        // Force cleanup of all IO bytes and explicit triggers on failure
        GVL.Robot.ACK_Complete     := 0;
        GVL.Robot.CMD              := 0;
        
        IF NOT xExecute THEN
            iHandshakeState := 0;
        END_IF;

END_CASE;

END_FUNCTION_BLOCK

// Device/Application/F002_PART_X/F002_SR01_SOCKET_SERVER
PROGRAM F002_SR01_SOCKET_SERVER
VAR
    ipAddr : NBS.IP_ADDR := (sAddr:= '192.168.0.247');
	Server: NBS.TCP_Server :=(uiPort :=2000);
	

	Connection: NBS.TCP_Connection;
	Read : NBS.TCP_Read;
	Write : NBS.TCP_Write;
	
	T1: TON := (PT := TIME#50MS);
	xEnableServer: BOOL;
	
	ReadData: ARRAY[0..3] OF DINT;
END_VAR
VAR_INPUT
	WriteData:  ARRAY[0..9] OF BYTE;
END_VAR

//TCP Sockets Server

//Server Instance
Server(xEnable:=GVL.PARTX.ENABLE_TCP,
		ipAddr:= ipAddr
		);
		
//Conection INstance	
Connection(xEnable:=(Server.xbusy AND NOT(Connection.xDone)),
		hServer:= Server.hServer
		);
		
//Read Data		
Read(xEnable:= Connection.xActive,
		hConnection:=Connection.hConnection,
		szSize:=SIZEOF(ReadData),
		pData:=ADR(ReadData)
		);

		
//Write Data	
Write(xExecute:= Connection.xActive AND T1.Q,
		hConnection:=Connection.hConnection,
		szSize:=SIZEOF(WriteData),
		pData:=ADR(WriteData)
		);

//Write Data Time Interval	
T1(IN:=NOT(Write.xDone));

END_PROGRAM

// Device/Application/F002_PART_X/F002_SR02_SOCKET_CLIENT
PROGRAM F002_SR02_SOCKET_CLIENT
VAR
    ipAddr : NBS.IP_ADDR := (sAddr:= '192.168.1.11');
	Client: NBS.TCP_Client :=(uiPort :=2000);
	

	Connection: NBS.TCP_Connection;
	Read : NBS.TCP_Read;
	Write : NBS.TCP_Write;
	
	T1: TON := (PT := TIME#50MS);
	xEnableServer: BOOL;
	
	ReadData: ARRAY[0..3] OF DINT;
END_VAR
VAR_INPUT
	WriteData:  ARRAY[0..9] OF BYTE;
END_VAR

//TCP Sockets Client

//Client Instance
Client(xEnable:=GVL.PARTX.ENABLE_TCP,
		ipAddr:= ipAddr
		);
		
		
//Read Data		
Read(xEnable:= Client.xActive,
		hConnection:=Client.hConnection,
		szSize:=SIZEOF(ReadData),
		pData:=ADR(ReadData)
		);

		
//Write Data	
Write(xExecute:= Client.xActive AND T1.Q,
		hConnection:=Client.hConnection,
		szSize:=SIZEOF(WriteData),
		pData:=ADR(WriteData)
		);

//Write Data Time Interval	
T1(IN:=NOT(Write.xDone));

END_PROGRAM

// Device/Application/F002_PART_X/F002_SR03_PARTX
PROGRAM F002_SR03_PARTX
VAR
END_VAR

(* body of a kind this reader does not render *)

METHOD BOUNCE : ARRAY[0..9]OF BYTE
VAR_INPUT
END_VAR
BOUNCE[0]:=30;
BOUNCE[1]:=30;
BOUNCE[2]:=30;
BOUNCE[3]:=30;
BOUNCE[4]:=45;
END_METHOD

METHOD CLEAR : ARRAY[0..9]OF BYTE
VAR_INPUT
END_VAR
CLEAR[0]:=0;
CLEAR[1]:=0;
CLEAR[2]:=0;
CLEAR[3]:=0;
CLEAR[4]:=0;
END_METHOD

METHOD IDLE : ARRAY[0..9]OF BYTE
VAR_INPUT
END_VAR
IDLE[0]:=0;
IDLE[1]:=0;
IDLE[2]:=0;
IDLE[3]:=0;
IDLE[4]:=0;
IDLE[5]:=0;
END_METHOD

METHOD IDLE_Trigger : ARRAY[0..9]OF BYTE
VAR_INPUT
END_VAR
IDLE_Trigger[0]:=0;
IDLE_Trigger[1]:=0;
IDLE_Trigger[2]:=0;
IDLE_Trigger[3]:=0;
IDLE_Trigger[4]:=0;
IDLE_Trigger[5]:=2;
END_METHOD

ACTION Manual_ACT:
IF GVL.PARTX.FWD THEN
	GVL.PARTX.IDLE:=FALSE;
END_IF

IF GVL.PARTX.REV THEN
	GVL.PARTX.IDLE:=FALSE;
END_IF
END_ACTION

METHOD MOVE_FWD : ARRAY[0..9]OF BYTE
VAR_INPUT
END_VAR
MOVE_FWD[0]:=30;
MOVE_FWD[1]:=30;
MOVE_FWD[2]:=0;
MOVE_FWD[3]:=0;
MOVE_FWD[4]:=60;
END_METHOD

METHOD MOVE_MANUAL : ARRAY[0..9]OF BYTE
VAR_INPUT
END_VAR
MOVE_MANUAL[0]:=GVL.PARTX.Amp1;
MOVE_MANUAL[1]:=GVL.PARTX.Amp2;
MOVE_MANUAL[2]:=GVL.PARTX.Amp3;
MOVE_MANUAL[3]:=GVL.PARTX.Amp4;
MOVE_MANUAL[4]:=GVL.PARTX.Freq;
IF GVL.PARTX.BackLight THEN
	MOVE_MANUAL[5].1:=1;
ELSE
	MOVE_MANUAL[5].1:=0;
END_IF
IF GVL.PARTX.Feeder_Enable THEN
	MOVE_MANUAL[5].3:=1;
ELSE
	MOVE_MANUAL[5].3:=0;
END_IF
MOVE_MANUAL[6]:=0;
MOVE_MANUAL[7]:=0;
MOVE_MANUAL[8]:=0;
MOVE_MANUAL[9]:=0;
END_METHOD

METHOD MOVE_REV : ARRAY[0..9]OF BYTE
VAR_INPUT
END_VAR
MOVE_REV[0]:=0;
MOVE_REV[1]:=0;
MOVE_REV[2]:=30;
MOVE_REV[3]:=30;
MOVE_REV[4]:=60;
END_METHOD

METHOD SCHED : ARRAY[0..9]OF BYTE
VAR
	PartX_DelayTimer : TON;
    
    // Edge Trigger to catch the exact moment SCHED turns ON
    SchedTrigger : R_TRIG; 
    
    // Reusable timer for step delays
    StateTimer   : TON;
END_VAR
IF GVL.PARTX.SCHED THEN
	GVL.PARTX.FWD := TRUE;
	
	PartX_DelayTimer(IN := GVL.PARTX.FWD, PT := T#500MS);
	
	IF PartX_DelayTimer.Q THEN
		GVL.PARTX.FWD := FALSE;
		GVL.PARTX.REV := TRUE;
	END_IF;
END_IF
END_METHOD

ACTION SCHED_ACT:
// 1. Run the system blocks using the shared parent variables
SchedTrigger(CLK := GVL.PARTX.SCHED);
StateTimer();

// 2. The Finite State Machine
CASE CurrentState OF

    E_SchedState.INIT:
        GVL.PARTX.FWD := FALSE;
        GVL.PARTX.REV := FALSE;
        StateTimer(IN := FALSE); 
        CurrentState := E_SchedState.WAIT_FOR_START;

    E_SchedState.WAIT_FOR_START:
		GVL.PARTX.FWD := FALSE;
        GVL.PARTX.REV := FALSE;
        IF SchedTrigger.Q THEN
            CurrentState := E_SchedState.RUN_FORWARD;
        END_IF;

    E_SchedState.RUN_FORWARD:
        GVL.PARTX.FWD := TRUE;
        StateTimer(IN := TRUE, PT := T#5000MS);
        
        IF StateTimer.Q THEN
            GVL.PARTX.FWD := FALSE;  
            StateTimer(IN := FALSE); 
            CurrentState := E_SchedState.RUN_REVERSE;
        END_IF;

    E_SchedState.RUN_REVERSE:
        GVL.PARTX.REV := TRUE;
        StateTimer(IN := TRUE, PT := T#5000MS);
        
        IF StateTimer.Q THEN
            GVL.PARTX.REV := FALSE;  
            StateTimer(IN := FALSE); 
            CurrentState := E_SchedState.DONE;
        END_IF;
		GVL.PARTX.SCHED:=FALSE;

    E_SchedState.DONE:
        CurrentState := E_SchedState.INIT;

END_CASE;
END_ACTION

END_PROGRAM

// Device/Application/F1000_FBs/Meca500/Delay
FUNCTION_BLOCK Delay
VAR_INPUT
	Seconds					:	REAL;
	ExternalStatecontrol 	:	BOOL;
	ExternalMoveID			:	UINT;
END_VAR
VAR_IN_OUT
	Robot	:	Meca500;	
	Sent		:	BOOL;
	Buffered	:	BOOL;
END_VAR
VAR_OUTPUT
	Error		:	BOOL;
END_VAR
VAR
	Output_Params	:	ARRAY[1..6] OF REAL;
	FirstScan: BOOL;
END_VAR

        (*Collect Inputs and store them locally*)
Output_Params[1]:=Seconds;
Output_Params[2]:=0;
Output_Params[3]:=0;
Output_Params[4]:=0;
Output_Params[5]:=0;
Output_Params[6]:=0;


(* If Values have change, Reinitialise Outputs*)

IF FirstScan=0 OR Robot.Outputs.MotionCommand.Argument0 <> Output_Params[1] OR Robot.Outputs.MotionCommand.Argument1 <> Output_Params[2] OR Robot.Outputs.MotionCommand.Argument2 <> Output_Params[3] OR Robot.Outputs.MotionCommand.Argument3 <> Output_Params[4] OR Robot.Outputs.MotionCommand.Argument4 <> Output_Params[5] OR Robot.Outputs.MotionCommand.Argument5 <> Output_Params[6] THEN
	Buffered := FALSE;
	Sent := FALSE;
END_IF;

(*if not in legacy mode, Act Setpoint*)
IF Robot.Outputs.MoveID <> 0 THEN
    Robot.Outputs.MotionControl.SetPoint := TRUE;
END_IF;

(* To send _Move, send _Move ID *)
IF NOT Buffered AND NOT Sent THEN
    
    Robot.Outputs.MotionCommand.MoveCommand := Meca500_MotionCommandID.DELAY;
    Robot.Outputs.MotionCommand.Argument0 := Output_Params[1];
	Robot.Outputs.MotionCommand.Argument1 := Output_Params[2];
	Robot.Outputs.MotionCommand.Argument2 := Output_Params[3];
	Robot.Outputs.MotionCommand.Argument3 := Output_Params[4];
	Robot.Outputs.MotionCommand.Argument4 := Output_Params[5];
	Robot.Outputs.MotionCommand.Argument5 := Output_Params[6];
    
    IF ExternalStateControl THEN
        IF ExternalMoveID <> 0 AND ExternalMoveID <> 32060 AND ExternalMoveID <> 32061 THEN
            Robot.Outputs.MoveID := ExternalMoveID;
            Sent := TRUE;
        END_IF;
        
    ELSE (*Not External Control*)
        IF Robot.Outputs.MoveID = 32060 THEN
            Robot.Outputs.MoveID := 32061;
        ELSIF Robot.Outputs.MoveID = 32061 THEN
            Robot.Outputs.MoveID := 32060;
        ELSIF Robot.Outputs.MoveID <> 32060 OR Robot.Outputs.MoveID <> 32061 THEN
            Robot.Outputs.MoveID := 32060;
        END_IF;
        Sent := TRUE;
    END_IF;
END_IF;

(* Check if _Move has been sent, if so, check if it was received *)
IF Sent THEN
    IF Robot.Outputs.MotionCommand.MoveCommand = Meca500_MotionCommandID.DELAY THEN
        IF Robot.Outputs.MotionCommand.Argument0 = Output_Params[1] AND Robot.Outputs.MotionCommand.Argument1 = Output_Params[2] AND Robot.Outputs.MotionCommand.Argument2 = Output_Params[3] AND Robot.Outputs.MotionCommand.Argument3 = Output_Params[4] AND Robot.Outputs.MotionCommand.Argument4 = Output_Params[5] AND Robot.Outputs.MotionCommand.Argument5 = Output_Params[6] THEN
            IF Robot.Inputs.Motion.MoveID = Robot.Outputs.MoveID THEN
                Buffered := TRUE;
            END_IF;
        END_IF;
    END_IF;
END_IF;

(*If External _Move ID is equal to Internal, raise an error*)
IF ExternalMoveID = 32060 OR ExternalMoveID = 32061 THEN
    Error := TRUE;
END_IF;
FirstScan := TRUE;

END_FUNCTION_BLOCK

// Device/Application/F1000_FBs/Meca500/GetErrors
FUNCTION_BLOCK GetErrors
VAR_INPUT
    RobotStatus_Error : UINT; // Mapped from Meca500_Inputs.RobotStatus_Error 
END_VAR

VAR_OUTPUT
    ErrorIsPresent : BOOL;
    CommandBufferFull : BOOL;
    UnknownCommand : BOOL;
    SyntaxError : BOOL;
    ArgumentError : BOOL;
    RobotNotActivated : BOOL;
    RobotNotHomed : BOOL;
    JointOverLimit : BOOL;
    LinearMoveBlockedByRotation : BOOL;
    RobotInError : BOOL;
    SingularityDetected : BOOL;
    ActivationFailed : BOOL;
    HomingFailed : BOOL;
    PoseOutOfReach : BOOL;
    CommunicationFailed : BOOL;
    MissingNULL : BOOL;
    BrakesError : BOOL;
    DeactivationFailed : BOOL;
    RobotNotSaving : BOOL;
    CommandNotExecutedInOfflineMode : BOOL;
    MasteringNeeded : BOOL;
    ImpossibleToReset : BOOL;
    DeactivationNeeded : BOOL;
    RobotMustBeDeactivated : BOOL;
    NetworkError : BOOL;
    MemoryFull : BOOL;
    AlreadySaving : BOOL;
    IsSaving : BOOL;
    StartConfMismatch : BOOL;
    GripperNotDetected : BOOL;
    CommandFailed : BOOL;
    NoVBox : BOOL;
    ExtToolSimMustDeact : BOOL;
    AnotherUserConnected : BOOL;
    CommandTooLong : BOOL;
    ErrorOfMotion : BOOL;
    DriveError : BOOL;
    InitializationFailed : BOOL;
    ErrorSaving : BOOL;
    InvalidOfflineProgram : BOOL;
    GripperError : BOOL;
    HardwareProblem : BOOL;
    ExcessiveTorque : BOOL;
    PneumaticError : BOOL;
    ExtToolNeedUpdate : BOOL;
    ImminentCollision : BOOL;
    IoPortPacketLost : BOOL;
    IoPortCommError : BOOL;
    ImminentCollisionDetected : BOOL;
    FailToMountDrive : BOOL;
    AtWorkZoneLimit : BOOL;
END_VAR

(* Logic Implementation *)
// Rung 0: General Error Check 
ErrorIsPresent := (RobotStatus_Error <> 0);

// Rungs 1-50: Specific Error Code Mapping [cite: 42, 43, 44, 45, 46, 47, 48, 49, 50, 51, 52, 53, 55, 56, 59, 60, 61, 63, 64]
CommandBufferFull := (RobotStatus_Error = 1000);
UnknownCommand    := (RobotStatus_Error = 1001);
SyntaxError       := (RobotStatus_Error = 1002);
ArgumentError     := (RobotStatus_Error = 1003);
RobotNotActivated := (RobotStatus_Error = 1005);
RobotNotHomed     := (RobotStatus_Error = 1006);
JointOverLimit    := (RobotStatus_Error = 1007);
LinearMoveBlockedByRotation := (RobotStatus_Error = 1010);
RobotInError      := (RobotStatus_Error = 1011);
SingularityDetected := (RobotStatus_Error = 1012);
ActivationFailed   := (RobotStatus_Error = 1013);
HomingFailed       := (RobotStatus_Error = 1014);
PoseOutOfReach     := (RobotStatus_Error = 1016);
CommunicationFailed := (RobotStatus_Error = 1017);
MissingNULL        := (RobotStatus_Error = 1018);
BrakesError        := (RobotStatus_Error = 1020);
DeactivationFailed := (RobotStatus_Error = 1021);
RobotNotSaving     := (RobotStatus_Error = 1022);
CommandNotExecutedInOfflineMode := (RobotStatus_Error = 1023);
MasteringNeeded    := (RobotStatus_Error = 1024);
ImpossibleToReset  := (RobotStatus_Error = 1025);
DeactivationNeeded := (RobotStatus_Error = 1026);
RobotMustBeDeactivated := (RobotStatus_Error = 1027);
NetworkError       := (RobotStatus_Error = 1028);
MemoryFull         := (RobotStatus_Error = 1029);
AlreadySaving      := (RobotStatus_Error = 1030);
IsSaving           := (RobotStatus_Error = 1031);
StartConfMismatch  := (RobotStatus_Error = 1033);
GripperNotDetected := (RobotStatus_Error = 1038);
CommandFailed      := (RobotStatus_Error = 1040);
NoVBox             := (RobotStatus_Error = 1041);
ExtToolSimMustDeact := (RobotStatus_Error = 1042);
AnotherUserConnected := (RobotStatus_Error = 3001);
CommandTooLong     := (RobotStatus_Error = 3003);
ErrorOfMotion      := (RobotStatus_Error = 3005);
DriveError         := (RobotStatus_Error = 3006);
InitializationFailed := (RobotStatus_Error = 3009);
ErrorSaving        := (RobotStatus_Error = 3014);
InvalidOfflineProgram := (RobotStatus_Error = 3020);
GripperError       := (RobotStatus_Error = 3025);
HardwareProblem    := (RobotStatus_Error = 3026);
ExcessiveTorque    := (RobotStatus_Error = 3029);
PneumaticError     := (RobotStatus_Error = 3037);
ExtToolNeedUpdate  := (RobotStatus_Error = 3039);
ImminentCollision  := (RobotStatus_Error = 3041);
IoPortPacketLost   := (RobotStatus_Error = 3043);
IoPortCommError    := (RobotStatus_Error = 3044);
ImminentCollisionDetected := (RobotStatus_Error = 3045);
FailToMountDrive   := (RobotStatus_Error = 3047);
AtWorkZoneLimit    := (RobotStatus_Error = 3049);

END_FUNCTION_BLOCK

// Device/Application/F1000_FBs/Meca500/Gripper
FUNCTION_BLOCK Gripper
VAR_INPUT
	Open					:	REAL;
	ExternalStatecontrol 	:	BOOL;
	ExternalMoveID			:	UINT;
END_VAR
VAR_IN_OUT
	Robot	:	Meca500;	
	Sent		:	BOOL;
	Buffered	:	BOOL;
END_VAR
VAR_OUTPUT
	Error		:	BOOL;
END_VAR
VAR
	Output_Params	:	ARRAY[1..6] OF REAL;
	FirstScan: BOOL;
END_VAR

        (*Collect Inputs and store them locally*)
Output_Params[1]:=Open;
Output_Params[2]:=0;
Output_Params[3]:=0;
Output_Params[4]:=0;
Output_Params[5]:=0;
Output_Params[6]:=0;


(* If Values have change, Reinitialise Outputs*)

IF FirstScan=0 OR Robot.Outputs.MotionCommand.Argument0 <> Output_Params[1] OR Robot.Outputs.MotionCommand.Argument1 <> Output_Params[2] OR Robot.Outputs.MotionCommand.Argument2 <> Output_Params[3] OR Robot.Outputs.MotionCommand.Argument3 <> Output_Params[4] OR Robot.Outputs.MotionCommand.Argument4 <> Output_Params[5] OR Robot.Outputs.MotionCommand.Argument5 <> Output_Params[6] THEN
	Buffered := FALSE;
	Sent := FALSE;
END_IF;

(*if not in legacy mode, Act Setpoint*)
IF Robot.Outputs.MoveID <> 0 THEN
    Robot.Outputs.MotionControl.SetPoint := TRUE;
END_IF;

(* To send _Move, send _Move ID *)
IF NOT Buffered AND NOT Sent THEN
    
    Robot.Outputs.MotionCommand.MoveCommand := Meca500_MotionCommandID.GRIPPER;
    Robot.Outputs.MotionCommand.Argument0 := Output_Params[1];
	Robot.Outputs.MotionCommand.Argument1 := Output_Params[2];
	Robot.Outputs.MotionCommand.Argument2 := Output_Params[3];
	Robot.Outputs.MotionCommand.Argument3 := Output_Params[4];
	Robot.Outputs.MotionCommand.Argument4 := Output_Params[5];
	Robot.Outputs.MotionCommand.Argument5 := Output_Params[6];
    
    IF ExternalStateControl THEN
        IF ExternalMoveID <> 0 AND ExternalMoveID <> 32180 AND ExternalMoveID <> 32181 THEN
            Robot.Outputs.MoveID := ExternalMoveID;
            Sent := TRUE;
        END_IF;
        
    ELSE (*Not External Control*)
        IF Robot.Outputs.MoveID = 32180 THEN
            Robot.Outputs.MoveID := 32181;
        ELSIF Robot.Outputs.MoveID = 32181 THEN
            Robot.Outputs.MoveID := 32180;
        ELSIF Robot.Outputs.MoveID <> 32180 OR Robot.Outputs.MoveID <> 32181 THEN
            Robot.Outputs.MoveID := 32180;
        END_IF;
        Sent := TRUE;
    END_IF;
END_IF;

(* Check if _Move has been sent, if so, check if it was received *)
IF Sent THEN
    IF Robot.Outputs.MotionCommand.MoveCommand = Meca500_MotionCommandID.GRIPPER THEN
        IF Robot.Outputs.MotionCommand.Argument0 = Output_Params[1] AND Robot.Outputs.MotionCommand.Argument1 = Output_Params[2] AND Robot.Outputs.MotionCommand.Argument2 = Output_Params[3] AND Robot.Outputs.MotionCommand.Argument3 = Output_Params[4] AND Robot.Outputs.MotionCommand.Argument4 = Output_Params[5] AND Robot.Outputs.MotionCommand.Argument5 = Output_Params[6] THEN
            IF Robot.Inputs.Motion.MoveID = Robot.Outputs.MoveID THEN
                Buffered := TRUE;
            END_IF;
        END_IF;
    END_IF;
END_IF;

(*If External _Move ID is equal to Internal, raise an error*)
IF ExternalMoveID = 32180 OR ExternalMoveID = 32181 THEN
    Error := TRUE;
END_IF;
FirstScan := TRUE;

END_FUNCTION_BLOCK

// Device/Application/F1000_FBs/Meca500/MoveGripper
FUNCTION_BLOCK MoveGripper
VAR_INPUT
	mm				:	REAL;
	ExternalStatecontrol 	:	BOOL;
	ExternalMoveID			:	UINT;
END_VAR
VAR_IN_OUT
	Robot	:	Meca500;	
	Sent		:	BOOL;
	Buffered	:	BOOL;
END_VAR
VAR_OUTPUT
	Error		:	BOOL;
END_VAR
VAR
	Output_Params	:	ARRAY[1..6] OF REAL;
	FirstScan: BOOL;
END_VAR

        (*Collect Inputs and store them locally*)
Output_Params[1]:=mm;
Output_Params[2]:=0;
Output_Params[3]:=0;
Output_Params[4]:=0;
Output_Params[5]:=0;
Output_Params[6]:=0;


(* If Values have change, Reinitialise Outputs*)

IF FirstScan=0 OR Robot.Outputs.MotionCommand.Argument0 <> Output_Params[1] OR Robot.Outputs.MotionCommand.Argument1 <> Output_Params[2] OR Robot.Outputs.MotionCommand.Argument2 <> Output_Params[3] OR Robot.Outputs.MotionCommand.Argument3 <> Output_Params[4] OR Robot.Outputs.MotionCommand.Argument4 <> Output_Params[5] OR Robot.Outputs.MotionCommand.Argument5 <> Output_Params[6] THEN
	Buffered := FALSE;
	Sent := FALSE;
END_IF;


(*if not in legacy mode, Act Setpoint*)
IF Robot.Outputs.MoveID <> 0 THEN
    Robot.Outputs.MotionControl.SetPoint := TRUE;
END_IF;

(* To send _Move, send _Move ID *)
IF NOT Buffered AND NOT Sent THEN
    
    Robot.Outputs.MotionCommand.MoveCommand := Meca500_MotionCommandID.MOVE_GRIPPER;
    Robot.Outputs.MotionCommand.Argument0 := Output_Params[1];
	Robot.Outputs.MotionCommand.Argument1 := Output_Params[2];
	Robot.Outputs.MotionCommand.Argument2 := Output_Params[3];
	Robot.Outputs.MotionCommand.Argument3 := Output_Params[4];
	Robot.Outputs.MotionCommand.Argument4 := Output_Params[5];
	Robot.Outputs.MotionCommand.Argument5 := Output_Params[6];
    
    IF ExternalStateControl THEN
        IF ExternalMoveID <> 0 AND ExternalMoveID <> 32320 AND ExternalMoveID <> 32321 THEN
            Robot.Outputs.MoveID := ExternalMoveID;
            Sent := TRUE;
        END_IF;
        
    ELSE (*Not External Control*)
        IF Robot.Outputs.MoveID = 32320 THEN
            Robot.Outputs.MoveID := 32321;
        ELSIF Robot.Outputs.MoveID = 32321 THEN
            Robot.Outputs.MoveID := 32320;
        ELSIF Robot.Outputs.MoveID <> 32320 OR Robot.Outputs.MoveID <> 32321 THEN
            Robot.Outputs.MoveID := 32320;
        END_IF;
        Sent := TRUE;
    END_IF;
END_IF;

(* Check if _Move has been sent, if so, check if it was received *)
IF Sent THEN
    IF Robot.Outputs.MotionCommand.MoveCommand = Meca500_MotionCommandID.Move_GRIPPER THEN
        IF Robot.Outputs.MotionCommand.Argument0 = Output_Params[1] AND Robot.Outputs.MotionCommand.Argument1 = Output_Params[2] AND Robot.Outputs.MotionCommand.Argument2 = Output_Params[3] AND Robot.Outputs.MotionCommand.Argument3 = Output_Params[4] AND Robot.Outputs.MotionCommand.Argument4 = Output_Params[5] AND Robot.Outputs.MotionCommand.Argument5 = Output_Params[6] THEN
            IF Robot.Inputs.Motion.MoveID = Robot.Outputs.MoveID THEN
                Buffered := TRUE;
            END_IF;
        END_IF;
    END_IF;
END_IF;

(*If External _Move ID is equal to Internal, raise an error*)
IF ExternalMoveID = 32320 OR ExternalMoveID = 32321 THEN
    Error := TRUE;
END_IF;
FirstScan := TRUE;

END_FUNCTION_BLOCK

// Device/Application/F1000_FBs/Meca500/MoveJointsRel
FUNCTION_BLOCK MoveJointsRel
VAR_INPUT
	Joint_Angle				:	ARRAY[1..6]OF REAL;
	ExternalStatecontrol 	:	BOOL;
	ExternalMoveID			:	UINT;
END_VAR
VAR_IN_OUT
	Robot	:	Meca500;	
	Sent		:	BOOL:=0;
	Buffered	:	BOOL:=0;
END_VAR
VAR_OUTPUT
	Error		:	BOOL;
END_VAR
VAR
	{attribute 'initialize_on_call'}
	FirstScan: BOOL:=0;
	Output_Params	:	ARRAY[1..6] OF REAL;
	
END_VAR


        (*Collect Inputs and store them locally*)
Output_Params[1]:=Joint_Angle[1];
Output_Params[2]:=Joint_Angle[2];
Output_Params[3]:=Joint_Angle[3];
Output_Params[4]:=Joint_Angle[4];
Output_Params[5]:=Joint_Angle[5];
Output_Params[6]:=Joint_Angle[6];


(* If Values have change, Reinitialise Outputs*)

IF FirstScan=0 OR Robot.Outputs.MotionCommand.Argument0 <> Output_Params[1] OR Robot.Outputs.MotionCommand.Argument1 <> Output_Params[2] OR Robot.Outputs.MotionCommand.Argument2 <> Output_Params[3] OR Robot.Outputs.MotionCommand.Argument3 <> Output_Params[4] OR Robot.Outputs.MotionCommand.Argument4 <> Output_Params[5] OR Robot.Outputs.MotionCommand.Argument5 <> Output_Params[6] THEN
	Buffered := FALSE;
	Sent := FALSE;
END_IF;


(*if not in legacy mode, Act Setpoint*)
IF Robot.Outputs.MoveID <> 0 THEN
    Robot.Outputs.MotionControl.SetPoint := TRUE;
END_IF;

(* To send _Move, send _Move ID *)
IF NOT Buffered AND NOT Sent THEN
    
    Robot.Outputs.MotionCommand.MoveCommand := Meca500_MotionCommandID.MOVE_JOINTS_REL;
    Robot.Outputs.MotionCommand.Argument0 := Output_Params[1];
	Robot.Outputs.MotionCommand.Argument1 := Output_Params[2];
	Robot.Outputs.MotionCommand.Argument2 := Output_Params[3];
	Robot.Outputs.MotionCommand.Argument3 := Output_Params[4];
	Robot.Outputs.MotionCommand.Argument4 := Output_Params[5];
	Robot.Outputs.MotionCommand.Argument5 := Output_Params[6];
    
    IF ExternalStateControl THEN
        IF ExternalMoveID <> 0 AND ExternalMoveID <> 32290 AND ExternalMoveID <> 32291 THEN
            Robot.Outputs.MoveID := ExternalMoveID;
            Sent := TRUE;
        END_IF;
        
    ELSE (*Not External Control*)
        IF Robot.Outputs.MoveID = 32290 THEN
            Robot.Outputs.MoveID := 32291;
        ELSIF Robot.Outputs.MoveID = 32291 THEN
            Robot.Outputs.MoveID := 32290;
        ELSIF Robot.Outputs.MoveID <> 32290 OR Robot.Outputs.MoveID <> 32291 THEN
            Robot.Outputs.MoveID := 32290;
        END_IF;
        Sent := TRUE;
    END_IF;
END_IF;

(* Check if _Move has been sent, if so, check if it was received *)
IF Sent THEN
    IF Robot.Outputs.MotionCommand.MoveCommand = Meca500_MotionCommandID.Move_JOINTS_REL THEN
        IF Robot.Outputs.MotionCommand.Argument0 = Output_Params[1] AND Robot.Outputs.MotionCommand.Argument1 = Output_Params[2] AND Robot.Outputs.MotionCommand.Argument2 = Output_Params[3] AND Robot.Outputs.MotionCommand.Argument3 = Output_Params[4] AND Robot.Outputs.MotionCommand.Argument4 = Output_Params[5] AND Robot.Outputs.MotionCommand.Argument5 = Output_Params[6] THEN
            IF Robot.Inputs.Motion.MoveID = Robot.Outputs.MoveID THEN
                Buffered := TRUE;
            END_IF;
        END_IF;
    END_IF;
END_IF;

(*If External _Move ID is equal to Internal, raise an error*)
IF ExternalMoveID = 32290 OR ExternalMoveID = 32291 THEN
    Error := TRUE;
END_IF;

FirstScan := TRUE;

END_FUNCTION_BLOCK

// Device/Application/F1000_FBs/Meca500/MoveJointsVel
FUNCTION_BLOCK MoveJointsVel
VAR_INPUT
	Joint_Velocity				:	ARRAY[1..6]OF REAL;
	ExternalStatecontrol 	:	BOOL;
	ExternalMoveID			:	UINT;
END_VAR
VAR_IN_OUT
	Robot	:	Meca500;	
	Sent		:	BOOL;
	Buffered	:	BOOL;
END_VAR
VAR_OUTPUT
	Error		:	BOOL;
END_VAR
VAR
	Output_Params	:	ARRAY[1..6] OF REAL;
	FirstScan: BOOL;

END_VAR

 
       (*Collect Inputs and store them locally*)
Output_Params[1]:=Joint_Velocity[1];
Output_Params[2]:=Joint_Velocity[2];
Output_Params[3]:=Joint_Velocity[3];
Output_Params[4]:=Joint_Velocity[4];
Output_Params[5]:=Joint_Velocity[5];
Output_Params[6]:=Joint_Velocity[6];


(* If Values have change, Reinitialise Outputs*)
    IF FirstScan=0 OR Robot.Outputs.MotionCommand.Argument0 <> Output_Params[1] OR Robot.Outputs.MotionCommand.Argument1 <> Output_Params[2] OR Robot.Outputs.MotionCommand.Argument2 <> Output_Params[3] OR Robot.Outputs.MotionCommand.Argument3 <> Output_Params[4] OR Robot.Outputs.MotionCommand.Argument4 <> Output_Params[5] OR Robot.Outputs.MotionCommand.Argument5 <> Output_Params[6] THEN
		Buffered := FALSE;
		Sent := FALSE;
	END_IF;


(*if not in legacy mode, Act Setpoint*)
IF Robot.Outputs.MoveID <> 0 THEN
    Robot.Outputs.MotionControl.SetPoint := TRUE;
END_IF;

(* To send _Move, send _Move ID *)
IF NOT Buffered AND NOT Sent THEN
    
    Robot.Outputs.MotionCommand.MoveCommand := Meca500_MotionCommandID.MOVE_JOINTS_VEL;
    Robot.Outputs.MotionCommand.Argument0 := Output_Params[1];
	Robot.Outputs.MotionCommand.Argument1 := Output_Params[2];
	Robot.Outputs.MotionCommand.Argument2 := Output_Params[3];
	Robot.Outputs.MotionCommand.Argument3 := Output_Params[4];
	Robot.Outputs.MotionCommand.Argument4 := Output_Params[5];
	Robot.Outputs.MotionCommand.Argument5 := Output_Params[6];
    
    IF ExternalStateControl THEN
        IF ExternalMoveID <> 0 AND ExternalMoveID <> 32210 AND ExternalMoveID <> 32211 THEN
            Robot.Outputs.MoveID := ExternalMoveID;
            Sent := TRUE;
        END_IF;
        
    ELSE (*Not External Control*)
        IF Robot.Outputs.MoveID = 32210 THEN
            Robot.Outputs.MoveID := 32211;
        ELSIF Robot.Outputs.MoveID = 32211 THEN
            Robot.Outputs.MoveID := 32210;
        ELSIF Robot.Outputs.MoveID <> 32210 OR Robot.Outputs.MoveID <> 32211 THEN
            Robot.Outputs.MoveID := 32210;
        END_IF;
        Sent := TRUE;
    END_IF;
END_IF;

(* Check if _Move has been sent, if so, check if it was received *)
IF Sent THEN
    IF Robot.Outputs.MotionCommand.MoveCommand = Meca500_MotionCommandID.Move_JOINTS_VEL THEN
        IF Robot.Outputs.MotionCommand.Argument0 = Output_Params[1] AND Robot.Outputs.MotionCommand.Argument1 = Output_Params[2] AND Robot.Outputs.MotionCommand.Argument2 = Output_Params[3] AND Robot.Outputs.MotionCommand.Argument3 = Output_Params[4] AND Robot.Outputs.MotionCommand.Argument4 = Output_Params[5] AND Robot.Outputs.MotionCommand.Argument5 = Output_Params[6] THEN
            IF Robot.Inputs.Motion.MoveID = Robot.Outputs.MoveID THEN
                Buffered := TRUE;
            END_IF;
        END_IF;
    END_IF;
END_IF;

(*If External _Move ID is equal to Internal, raise an error*)
IF ExternalMoveID = 32210 OR ExternalMoveID = 32211 THEN
    Error := TRUE;
END_IF;
FirstScan := TRUE;

END_FUNCTION_BLOCK

// Device/Application/F1000_FBs/Meca500/MoveLinRelWrf
FUNCTION_BLOCK MoveLinRelWrf
VAR_INPUT
	Pose					:	ARRAY[1..6]OF REAL;
	ExternalStatecontrol 	:	BOOL;
	ExternalMoveID			:	UINT;
END_VAR
VAR_IN_OUT
	Robot	:	Meca500;	
	Sent		:	BOOL;
	Buffered	:	BOOL;
END_VAR
VAR_OUTPUT
	Error		:	BOOL;
END_VAR
VAR
	Output_Params	:	ARRAY[1..6] OF REAL;
	FirstScan: BOOL;
END_VAR

        (*Collect Inputs and store them locally*)
Output_Params[1]:=Pose[1];
Output_Params[2]:=Pose[2];
Output_Params[3]:=Pose[3];
Output_Params[4]:=Pose[4];
Output_Params[5]:=Pose[5];
Output_Params[6]:=Pose[6];


(* If Values have change, Reinitialise Outputs*)

    IF FirstScan=0 OR Robot.Outputs.MotionCommand.Argument0 <> Output_Params[1] OR Robot.Outputs.MotionCommand.Argument1 <> Output_Params[2] OR Robot.Outputs.MotionCommand.Argument2 <> Output_Params[3] OR Robot.Outputs.MotionCommand.Argument3 <> Output_Params[4] OR Robot.Outputs.MotionCommand.Argument4 <> Output_Params[5] OR Robot.Outputs.MotionCommand.Argument5 <> Output_Params[6] THEN
		Buffered := FALSE;
		Sent := FALSE;
	END_IF;

(*if not in legacy mode, Act Setpoint*)
IF Robot.Outputs.MoveID <> 0 THEN
    Robot.Outputs.MotionControl.SetPoint := TRUE;
END_IF;

(* To send _Move, send _Move ID *)
IF NOT Buffered AND NOT Sent THEN
    
    Robot.Outputs.MotionCommand.MoveCommand := Meca500_MotionCommandID.MOVE_LIN_REL_WRF;
    Robot.Outputs.MotionCommand.Argument0 := Output_Params[1];
	Robot.Outputs.MotionCommand.Argument1 := Output_Params[2];
	Robot.Outputs.MotionCommand.Argument2 := Output_Params[3];
	Robot.Outputs.MotionCommand.Argument3 := Output_Params[4];
	Robot.Outputs.MotionCommand.Argument4 := Output_Params[5];
	Robot.Outputs.MotionCommand.Argument5 := Output_Params[6];
    
    IF ExternalStateControl THEN
        IF ExternalMoveID <> 0 AND ExternalMoveID <> 32050 AND ExternalMoveID <> 32051 THEN
            Robot.Outputs.MoveID := ExternalMoveID;
            Sent := TRUE;
        END_IF;
        
    ELSE (*Not External Control*)
        IF Robot.Outputs.MoveID = 32050 THEN
            Robot.Outputs.MoveID := 32051;
        ELSIF Robot.Outputs.MoveID = 32051 THEN
            Robot.Outputs.MoveID := 32050;
        ELSIF Robot.Outputs.MoveID <> 32050 OR Robot.Outputs.MoveID <> 32051 THEN
            Robot.Outputs.MoveID := 32050;
        END_IF;
        Sent := TRUE;
    END_IF;
END_IF;

(* Check if _Move has been sent, if so, check if it was received *)
IF Sent THEN
    IF Robot.Outputs.MotionCommand.MoveCommand = Meca500_MotionCommandID.Move_LIN_REL_WRF THEN
        IF Robot.Outputs.MotionCommand.Argument0 = Output_Params[1] AND Robot.Outputs.MotionCommand.Argument1 = Output_Params[2] AND Robot.Outputs.MotionCommand.Argument2 = Output_Params[3] AND Robot.Outputs.MotionCommand.Argument3 = Output_Params[4] AND Robot.Outputs.MotionCommand.Argument4 = Output_Params[5] AND Robot.Outputs.MotionCommand.Argument5 = Output_Params[6] THEN
            IF Robot.Inputs.Motion.MoveID = Robot.Outputs.MoveID THEN
                Buffered := TRUE;
            END_IF;
        END_IF;
    END_IF;
END_IF;

(*If External _Move ID is equal to Internal, raise an error*)
IF ExternalMoveID = 32050 OR ExternalMoveID = 32051 THEN
    Error := TRUE;
END_IF;
FirstScan := TRUE;

END_FUNCTION_BLOCK

// Device/Application/F1000_FBs/Meca500/MoveLinVelTrf
FUNCTION_BLOCK MoveLinVelTrf
VAR_INPUT
	Velocity					:	ARRAY[1..6]OF REAL;
	ExternalStatecontrol 	:	BOOL;
	ExternalMoveID			:	UINT;
END_VAR
VAR_IN_OUT
	Robot	:	Meca500;	
	Sent		:	BOOL;
	Buffered	:	BOOL;
END_VAR
VAR_OUTPUT
	Error		:	BOOL;
END_VAR
VAR
	Output_Params	:	ARRAY[1..6] OF REAL;
	FirstScan: BOOL;
END_VAR

        (*Collect Inputs and store them locally*)
Output_Params[1]:=Velocity[1];
Output_Params[2]:=Velocity[2];
Output_Params[3]:=Velocity[3];
Output_Params[4]:=Velocity[4];
Output_Params[5]:=Velocity[5];
Output_Params[6]:=Velocity[6];


(* If Values have change, Reinitialise Outputs*)

IF FirstScan=0 OR Robot.Outputs.MotionCommand.Argument0 <> Output_Params[1] OR Robot.Outputs.MotionCommand.Argument1 <> Output_Params[2] OR Robot.Outputs.MotionCommand.Argument2 <> Output_Params[3] OR Robot.Outputs.MotionCommand.Argument3 <> Output_Params[4] OR Robot.Outputs.MotionCommand.Argument4 <> Output_Params[5] OR Robot.Outputs.MotionCommand.Argument5 <> Output_Params[6] THEN
	Buffered := FALSE;
	Sent := FALSE;
END_IF;


(*if not in legacy mode, Act Setpoint*)
IF Robot.Outputs.MoveID <> 0 THEN
    Robot.Outputs.MotionControl.SetPoint := TRUE;
END_IF;

(* To send _Move, send _Move ID *)
IF NOT Buffered AND NOT Sent THEN
    
    Robot.Outputs.MotionCommand.MoveCommand := Meca500_MotionCommandID.MOVE_LIN_VEL_TRF;
    Robot.Outputs.MotionCommand.Argument0 := Output_Params[1];
	Robot.Outputs.MotionCommand.Argument1 := Output_Params[2];
	Robot.Outputs.MotionCommand.Argument2 := Output_Params[3];
	Robot.Outputs.MotionCommand.Argument3 := Output_Params[4];
	Robot.Outputs.MotionCommand.Argument4 := Output_Params[5];
	Robot.Outputs.MotionCommand.Argument5 := Output_Params[6];
    
    IF ExternalStateControl THEN
        IF ExternalMoveID <> 0 AND ExternalMoveID <> 32230 AND ExternalMoveID <> 32231 THEN
            Robot.Outputs.MoveID := ExternalMoveID;
            Sent := TRUE;
        END_IF;
        
    ELSE (*Not External Control*)
        IF Robot.Outputs.MoveID = 32230 THEN
            Robot.Outputs.MoveID := 32231;
        ELSIF Robot.Outputs.MoveID = 32231 THEN
            Robot.Outputs.MoveID := 32230;
        ELSIF Robot.Outputs.MoveID <> 32230 OR Robot.Outputs.MoveID <> 32231 THEN
            Robot.Outputs.MoveID := 32230;
        END_IF;
        Sent := TRUE;
    END_IF;
END_IF;

(* Check if _Move has been sent, if so, check if it was received *)
IF Sent THEN
    IF Robot.Outputs.MotionCommand.MoveCommand = Meca500_MotionCommandID.Move_LIN_VEL_TRF THEN
        IF Robot.Outputs.MotionCommand.Argument0 = Output_Params[1] AND Robot.Outputs.MotionCommand.Argument1 = Output_Params[2] AND Robot.Outputs.MotionCommand.Argument2 = Output_Params[3] AND Robot.Outputs.MotionCommand.Argument3 = Output_Params[4] AND Robot.Outputs.MotionCommand.Argument4 = Output_Params[5] AND Robot.Outputs.MotionCommand.Argument5 = Output_Params[6] THEN
            IF Robot.Inputs.Motion.MoveID = Robot.Outputs.MoveID THEN
                Buffered := TRUE;
            END_IF;
        END_IF;
    END_IF;
END_IF;

(*If External _Move ID is equal to Internal, raise an error*)
IF ExternalMoveID = 32230 OR ExternalMoveID = 32231 THEN
    Error := TRUE;
END_IF;
FirstScan := TRUE;

END_FUNCTION_BLOCK

// Device/Application/F1000_FBs/Meca500/MoveLinVelWrf
FUNCTION_BLOCK MoveLinVelWrf
VAR_INPUT
	Velocity					:	ARRAY[1..6]OF REAL;
	ExternalStatecontrol 	:	BOOL;
	ExternalMoveID			:	UINT;
END_VAR
VAR_IN_OUT
	Robot	:	Meca500;	
	Sent		:	BOOL;
	Buffered	:	BOOL;
END_VAR
VAR_OUTPUT
	Error		:	BOOL;
END_VAR
VAR
	Output_Params	:	ARRAY[1..6] OF REAL;
	FirstScan: BOOL;
END_VAR

        (*Collect Inputs and store them locally*)
Output_Params[1]:=Velocity[1];
Output_Params[2]:=Velocity[2];
Output_Params[3]:=Velocity[3];
Output_Params[4]:=Velocity[4];
Output_Params[5]:=Velocity[5];
Output_Params[6]:=Velocity[6];


(* If Values have change, Reinitialise Outputs*)

IF FirstScan=0 OR Robot.Outputs.MotionCommand.Argument0 <> Output_Params[1] OR Robot.Outputs.MotionCommand.Argument1 <> Output_Params[2] OR Robot.Outputs.MotionCommand.Argument2 <> Output_Params[3] OR Robot.Outputs.MotionCommand.Argument3 <> Output_Params[4] OR Robot.Outputs.MotionCommand.Argument4 <> Output_Params[5] OR Robot.Outputs.MotionCommand.Argument5 <> Output_Params[6] THEN
	Buffered := FALSE;
	Sent := FALSE;
END_IF;


(*if not in legacy mode, Act Setpoint*)
IF Robot.Outputs.MoveID <> 0 THEN
    Robot.Outputs.MotionControl.SetPoint := TRUE;
END_IF;

(* To send _Move, send _Move ID *)
IF NOT Buffered AND NOT Sent THEN
    
    Robot.Outputs.MotionCommand.MoveCommand := Meca500_MotionCommandID.MOVE_LIN_VEL_WRF;
    Robot.Outputs.MotionCommand.Argument0 := Output_Params[1];
	Robot.Outputs.MotionCommand.Argument1 := Output_Params[2];
	Robot.Outputs.MotionCommand.Argument2 := Output_Params[3];
	Robot.Outputs.MotionCommand.Argument3 := Output_Params[4];
	Robot.Outputs.MotionCommand.Argument4 := Output_Params[5];
	Robot.Outputs.MotionCommand.Argument5 := Output_Params[6];
    
    IF ExternalStateControl THEN
        IF ExternalMoveID <> 0 AND ExternalMoveID <> 32220 AND ExternalMoveID <> 32221 THEN
            Robot.Outputs.MoveID := ExternalMoveID;
            Sent := TRUE;
        END_IF;
        
    ELSE (*Not External Control*)
        IF Robot.Outputs.MoveID = 32220 THEN
            Robot.Outputs.MoveID := 32221;
        ELSIF Robot.Outputs.MoveID = 32221 THEN
            Robot.Outputs.MoveID := 32220;
        ELSIF Robot.Outputs.MoveID <> 32220 OR Robot.Outputs.MoveID <> 32221 THEN
            Robot.Outputs.MoveID := 32220;
        END_IF;
        Sent := TRUE;
    END_IF;
END_IF;

(* Check if _Move has been sent, if so, check if it was received *)
IF Sent THEN
    IF Robot.Outputs.MotionCommand.MoveCommand = Meca500_MotionCommandID.Move_LIN_VEL_WRF THEN
        IF Robot.Outputs.MotionCommand.Argument0 = Output_Params[1] AND Robot.Outputs.MotionCommand.Argument1 = Output_Params[2] AND Robot.Outputs.MotionCommand.Argument2 = Output_Params[3] AND Robot.Outputs.MotionCommand.Argument3 = Output_Params[4] AND Robot.Outputs.MotionCommand.Argument4 = Output_Params[5] AND Robot.Outputs.MotionCommand.Argument5 = Output_Params[6] THEN
            IF Robot.Inputs.Motion.MoveID = Robot.Outputs.MoveID THEN
                Buffered := TRUE;
            END_IF;
        END_IF;
    END_IF;
END_IF;

(*If External _Move ID is equal to Internal, raise an error*)
IF ExternalMoveID = 32220 OR ExternalMoveID = 32221 THEN
    Error := TRUE;
END_IF;
FirstScan := TRUE;

END_FUNCTION_BLOCK

// Device/Application/F1000_FBs/Meca500/SetAutoConf
FUNCTION_BLOCK SetAutoConf
VAR_INPUT
	Enable					:	REAL;
	ExternalStatecontrol 	:	BOOL;
	ExternalMoveID			:	UINT;
END_VAR
VAR_IN_OUT
	Robot	:	Meca500;	
	Sent		:	BOOL;
	Buffered	:	BOOL;
END_VAR
VAR_OUTPUT
	Error		:	BOOL;
END_VAR
VAR
	Output_Params	:	ARRAY[1..6] OF REAL;
	FirstScan: BOOL;
END_VAR

        (*Collect Inputs and store them locally*)
Output_Params[1]:=Enable;
Output_Params[2]:=0;
Output_Params[3]:=0;
Output_Params[4]:=0;
Output_Params[5]:=0;
Output_Params[6]:=0;


(* If Values have change, Reinitialise Outputs*)

IF 	FirstScan=0 OR Robot.Outputs.MotionCommand.Argument0 <> Output_Params[1] OR Robot.Outputs.MotionCommand.Argument1 <> Output_Params[2] OR Robot.Outputs.MotionCommand.Argument2 <> Output_Params[3] OR Robot.Outputs.MotionCommand.Argument3 <> Output_Params[4] OR Robot.Outputs.MotionCommand.Argument4 <> Output_Params[5] OR Robot.Outputs.MotionCommand.Argument5 <> Output_Params[6] THEN
	Buffered := FALSE;
	Sent := FALSE;
END_IF;


(*if not in legacy mode, Act Setpoint*)
IF Robot.Outputs.MoveID <> 0 THEN
    Robot.Outputs.MotionControl.SetPoint := TRUE;
END_IF;

(* To send _Move, send _Move ID *)
IF NOT Buffered AND NOT Sent THEN
    
    Robot.Outputs.MotionCommand.MoveCommand := Meca500_MotionCommandID.SET_AUTO_CONF;
    Robot.Outputs.MotionCommand.Argument0 := Output_Params[1];
	Robot.Outputs.MotionCommand.Argument1 := Output_Params[2];
	Robot.Outputs.MotionCommand.Argument2 := Output_Params[3];
	Robot.Outputs.MotionCommand.Argument3 := Output_Params[4];
	Robot.Outputs.MotionCommand.Argument4 := Output_Params[5];
	Robot.Outputs.MotionCommand.Argument5 := Output_Params[6];
    
    IF ExternalStateControl THEN
        IF ExternalMoveID <> 0 AND ExternalMoveID <> 32160 AND ExternalMoveID <> 32161 THEN
            Robot.Outputs.MoveID := ExternalMoveID;
            Sent := TRUE;
        END_IF;
        
    ELSE (*Not External Control*)
        IF Robot.Outputs.MoveID = 32160 THEN
            Robot.Outputs.MoveID := 32161;
        ELSIF Robot.Outputs.MoveID = 32161 THEN
            Robot.Outputs.MoveID := 32160;
        ELSIF Robot.Outputs.MoveID <> 32160 OR Robot.Outputs.MoveID <> 32161 THEN
            Robot.Outputs.MoveID := 32160;
        END_IF;
        Sent := TRUE;
    END_IF;
END_IF;

(* Check if _Move has been sent, if so, check if it was received *)
IF Sent THEN
    IF Robot.Outputs.MotionCommand.MoveCommand = Meca500_MotionCommandID.SET_AUTO_CONF THEN
        IF Robot.Outputs.MotionCommand.Argument0 = Output_Params[1] AND Robot.Outputs.MotionCommand.Argument1 = Output_Params[2] AND Robot.Outputs.MotionCommand.Argument2 = Output_Params[3] AND Robot.Outputs.MotionCommand.Argument3 = Output_Params[4] AND Robot.Outputs.MotionCommand.Argument4 = Output_Params[5] AND Robot.Outputs.MotionCommand.Argument5 = Output_Params[6] THEN
            IF Robot.Inputs.Motion.MoveID = Robot.Outputs.MoveID THEN
                Buffered := TRUE;
            END_IF;
        END_IF;
    END_IF;
END_IF;

(*If External _Move ID is equal to Internal, raise an error*)
IF ExternalMoveID = 32160 OR ExternalMoveID = 32161 THEN
    Error := TRUE;
END_IF;
FirstScan := TRUE;

END_FUNCTION_BLOCK

// Device/Application/F1000_FBs/Meca500/SetAutoConfTurn
FUNCTION_BLOCK SetAutoConfTurn
VAR_INPUT
	Enable					:	REAL;
	ExternalStatecontrol 	:	BOOL;
	ExternalMoveID			:	UINT;
END_VAR
VAR_IN_OUT
	Robot	:	Meca500;	
	Sent		:	BOOL;
	Buffered	:	BOOL;
END_VAR
VAR_OUTPUT
	Error		:	BOOL;
END_VAR
VAR
	Output_Params	:	ARRAY[1..6] OF REAL;
	FirstScan:Bool;
END_VAR

        (*Collect Inputs and store them locally*)
Output_Params[1]:=Enable;
Output_Params[2]:=0;
Output_Params[3]:=0;
Output_Params[4]:=0;
Output_Params[5]:=0;
Output_Params[6]:=0;

(* If Values have change, Reinitialise Outputs*)

IF FirstScan=0 OR Robot.Outputs.MotionCommand.Argument0 <> Output_Params[1] OR Robot.Outputs.MotionCommand.Argument1 <> Output_Params[2] OR Robot.Outputs.MotionCommand.Argument2 <> Output_Params[3] OR Robot.Outputs.MotionCommand.Argument3 <> Output_Params[4] OR Robot.Outputs.MotionCommand.Argument4 <> Output_Params[5] OR Robot.Outputs.MotionCommand.Argument5 <> Output_Params[6] THEN
	Buffered := FALSE;
	Sent := FALSE;
END_IF;


(*if not in legacy mode, Act Setpoint*)
IF Robot.Outputs.MoveID <> 0 THEN
    Robot.Outputs.MotionControl.SetPoint := TRUE;
END_IF;

(* To send _Move, send _Move ID *)
IF NOT Buffered AND NOT Sent THEN
    
    Robot.Outputs.MotionCommand.MoveCommand := Meca500_MotionCommandID.SET_AUTO_CONF_TURN;
    Robot.Outputs.MotionCommand.Argument0 := Output_Params[1];
	Robot.Outputs.MotionCommand.Argument1 := Output_Params[2];
	Robot.Outputs.MotionCommand.Argument2 := Output_Params[3];
	Robot.Outputs.MotionCommand.Argument3 := Output_Params[4];
	Robot.Outputs.MotionCommand.Argument4 := Output_Params[5];
	Robot.Outputs.MotionCommand.Argument5 := Output_Params[6];
    
    IF ExternalStateControl THEN
        IF ExternalMoveID <> 0 AND ExternalMoveID <> 32260 AND ExternalMoveID <> 32261 THEN
            Robot.Outputs.MoveID := ExternalMoveID;
            Sent := TRUE;
        END_IF;
        
    ELSE (*Not External Control*)
        IF Robot.Outputs.MoveID = 32260 THEN
            Robot.Outputs.MoveID := 32261;
        ELSIF Robot.Outputs.MoveID = 32261 THEN
            Robot.Outputs.MoveID := 32260;
        ELSIF Robot.Outputs.MoveID <> 32260 OR Robot.Outputs.MoveID <> 32261 THEN
            Robot.Outputs.MoveID := 32260;
        END_IF;
        Sent := TRUE;
    END_IF;
END_IF;

(* Check if _Move has been sent, if so, check if it was received *)
IF Sent THEN
    IF Robot.Outputs.MotionCommand.MoveCommand = Meca500_MotionCommandID.SET_AUTO_CONF_TURN THEN
        IF Robot.Outputs.MotionCommand.Argument0 = Output_Params[1] AND Robot.Outputs.MotionCommand.Argument1 = Output_Params[2] AND Robot.Outputs.MotionCommand.Argument2 = Output_Params[3] AND Robot.Outputs.MotionCommand.Argument3 = Output_Params[4] AND Robot.Outputs.MotionCommand.Argument4 = Output_Params[5] AND Robot.Outputs.MotionCommand.Argument5 = Output_Params[6] THEN
            IF Robot.Inputs.Motion.MoveID = Robot.Outputs.MoveID THEN
                Buffered := TRUE;
            END_IF;
        END_IF;
    END_IF;
END_IF;

(*If External _Move ID is equal to Internal, raise an error*)
IF ExternalMoveID = 32260 OR ExternalMoveID = 32261 THEN
    Error := TRUE;
END_IF;
FirstScan:=TRUE;

END_FUNCTION_BLOCK

// Device/Application/F1000_FBs/Meca500/SetBlending
FUNCTION_BLOCK SetBlending
VAR_INPUT
	Blending_Percentage					:	REAL;
	ExternalStatecontrol 	:	BOOL;
	ExternalMoveID			:	UINT;
END_VAR
VAR_IN_OUT
	Robot	:	Meca500;	
	Sent		:	BOOL;
	Buffered	:	BOOL;
END_VAR
VAR_OUTPUT
	Error		:	BOOL;
END_VAR
VAR
	Output_Params	:	ARRAY[1..6] OF REAL;
	FirstScan:BOOL;
END_VAR

        (*Collect Inputs and store them locally*)
Output_Params[1]:=Blending_Percentage;
Output_Params[2]:=0;
Output_Params[3]:=0;
Output_Params[4]:=0;
Output_Params[5]:=0;
Output_Params[6]:=0;


(* If Values have change, Reinitialise Outputs*)

IF FirstScan=0 OR Robot.Outputs.MotionCommand.Argument0 <> Output_Params[1] OR Robot.Outputs.MotionCommand.Argument1 <> Output_Params[2] OR Robot.Outputs.MotionCommand.Argument2 <> Output_Params[3] OR Robot.Outputs.MotionCommand.Argument3 <> Output_Params[4] OR Robot.Outputs.MotionCommand.Argument4 <> Output_Params[5] OR Robot.Outputs.MotionCommand.Argument5 <> Output_Params[6] THEN
	Buffered := FALSE;
	Sent := FALSE;
END_IF;

(*if not in legacy mode, Act Setpoint*)
IF Robot.Outputs.MoveID <> 0 THEN
    Robot.Outputs.MotionControl.SetPoint := TRUE;
END_IF;

(* To send _Move, send _Move ID *)
IF NOT Buffered AND NOT Sent THEN
    
    Robot.Outputs.MotionCommand.MoveCommand := Meca500_MotionCommandID.SET_BLENDING;
    Robot.Outputs.MotionCommand.Argument0 := Output_Params[1];
	Robot.Outputs.MotionCommand.Argument1 := Output_Params[2];
	Robot.Outputs.MotionCommand.Argument2 := Output_Params[3];
	Robot.Outputs.MotionCommand.Argument3 := Output_Params[4];
	Robot.Outputs.MotionCommand.Argument4 := Output_Params[5];
	Robot.Outputs.MotionCommand.Argument5 := Output_Params[6];
    
    IF ExternalStateControl THEN
        IF ExternalMoveID <> 0 AND ExternalMoveID <> 32070 AND ExternalMoveID <> 32071 THEN
            Robot.Outputs.MoveID := ExternalMoveID;
            Sent := TRUE;
        END_IF;
        
    ELSE (*Not External Control*)
        IF Robot.Outputs.MoveID = 32070 THEN
            Robot.Outputs.MoveID := 32071;
        ELSIF Robot.Outputs.MoveID = 32071 THEN
            Robot.Outputs.MoveID := 32070;
        ELSIF Robot.Outputs.MoveID <> 32070 OR Robot.Outputs.MoveID <> 32071 THEN
            Robot.Outputs.MoveID := 32070;
        END_IF;
        Sent := TRUE;
    END_IF;
END_IF;

(* Check if _Move has been sent, if so, check if it was received *)
IF Sent THEN
    IF Robot.Outputs.MotionCommand.MoveCommand = Meca500_MotionCommandID.SET_BLENDING THEN
        IF Robot.Outputs.MotionCommand.Argument0 = Output_Params[1] AND Robot.Outputs.MotionCommand.Argument1 = Output_Params[2] AND Robot.Outputs.MotionCommand.Argument2 = Output_Params[3] AND Robot.Outputs.MotionCommand.Argument3 = Output_Params[4] AND Robot.Outputs.MotionCommand.Argument4 = Output_Params[5] AND Robot.Outputs.MotionCommand.Argument5 = Output_Params[6] THEN
            IF Robot.Inputs.Motion.MoveID = Robot.Outputs.MoveID THEN
                Buffered := TRUE;
            END_IF;
        END_IF;
    END_IF;
END_IF;

(*If External _Move ID is equal to Internal, raise an error*)
IF ExternalMoveID = 32070 OR ExternalMoveID = 32071 THEN
    Error := TRUE;
END_IF;
FirstScan:=TRUE;

END_FUNCTION_BLOCK

// Device/Application/F1000_FBs/Meca500/SetCartAcc
FUNCTION_BLOCK SetCartAcc
VAR_INPUT
	Acceleration_Percentage					:	REAL;
	ExternalStatecontrol 	:	BOOL;
	ExternalMoveID			:	UINT;
END_VAR
VAR_IN_OUT
	Robot		:	Meca500;	
	Sent		:	BOOL;
	Buffered	:	BOOL;
END_VAR
VAR_OUTPUT
	Error		:	BOOL;
END_VAR
VAR
	Output_Params	:	ARRAY[1..6] OF REAL;
	FirstScan		:	BOOL;
END_VAR

        (*Collect Inputs and store them locally*)
Output_Params[1]:=Acceleration_Percentage;
Output_Params[2]:=0;
Output_Params[3]:=0;
Output_Params[4]:=0;
Output_Params[5]:=0;
Output_Params[6]:=0;


(* If Values have change, Reinitialise Outputs*)

IF FirstScan=0 OR Robot.Outputs.MotionCommand.Argument0 <> Output_Params[1] OR Robot.Outputs.MotionCommand.Argument1 <> Output_Params[2] OR Robot.Outputs.MotionCommand.Argument2 <> Output_Params[3] OR Robot.Outputs.MotionCommand.Argument3 <> Output_Params[4] OR Robot.Outputs.MotionCommand.Argument4 <> Output_Params[5] OR Robot.Outputs.MotionCommand.Argument5 <> Output_Params[6] THEN
	Buffered := FALSE;
	Sent := FALSE;
END_IF;

(*if not in legacy mode, Act Setpoint*)
IF Robot.Outputs.MoveID <> 0 THEN
    Robot.Outputs.MotionControl.SetPoint := TRUE;
END_IF;

(* To send _Move, send _Move ID *)
IF NOT Buffered AND NOT Sent THEN
    
    Robot.Outputs.MotionCommand.MoveCommand := Meca500_MotionCommandID.SET_CART_ACC;
    Robot.Outputs.MotionCommand.Argument0 := Output_Params[1];
	Robot.Outputs.MotionCommand.Argument1 := Output_Params[2];
	Robot.Outputs.MotionCommand.Argument2 := Output_Params[3];
	Robot.Outputs.MotionCommand.Argument3 := Output_Params[4];
	Robot.Outputs.MotionCommand.Argument4 := Output_Params[5];
	Robot.Outputs.MotionCommand.Argument5 := Output_Params[6];
    
    IF ExternalStateControl THEN
        IF ExternalMoveID <> 0 AND ExternalMoveID <> 32120 AND ExternalMoveID <> 32121 THEN
            Robot.Outputs.MoveID := ExternalMoveID;
            Sent := TRUE;
        END_IF;
        
    ELSE (*Not External Control*)
        IF Robot.Outputs.MoveID = 32120 THEN
            Robot.Outputs.MoveID := 32121;
        ELSIF Robot.Outputs.MoveID = 32121 THEN
            Robot.Outputs.MoveID := 32120;
        ELSIF Robot.Outputs.MoveID <> 32120 OR Robot.Outputs.MoveID <> 32121 THEN
            Robot.Outputs.MoveID := 32120;
        END_IF;
        Sent := TRUE;
    END_IF;
END_IF;

(* Check if _Move has been sent, if so, check if it was received *)
IF Sent THEN
    IF Robot.Outputs.MotionCommand.MoveCommand = Meca500_MotionCommandID.SET_CART_ACC THEN
        IF Robot.Outputs.MotionCommand.Argument0 = Output_Params[1] AND Robot.Outputs.MotionCommand.Argument1 = Output_Params[2] AND Robot.Outputs.MotionCommand.Argument2 = Output_Params[3] AND Robot.Outputs.MotionCommand.Argument3 = Output_Params[4] AND Robot.Outputs.MotionCommand.Argument4 = Output_Params[5] AND Robot.Outputs.MotionCommand.Argument5 = Output_Params[6] THEN
            IF Robot.Inputs.Motion.MoveID = Robot.Outputs.MoveID THEN
                Buffered := TRUE;
            END_IF;
        END_IF;
    END_IF;
END_IF;

(*If External _Move ID is equal to Internal, raise an error*)
IF ExternalMoveID = 32120 OR ExternalMoveID = 32121 THEN
    Error := TRUE;
END_IF;
FirstScan:=TRUE;

END_FUNCTION_BLOCK

// Device/Application/F1000_FBs/Meca500/SetCartAngVel
FUNCTION_BLOCK SetCartAngVel
VAR_INPUT
	Velocity_Limit					:	REAL;
	ExternalStatecontrol 	:	BOOL;
	ExternalMoveID			:	UINT;
END_VAR
VAR_IN_OUT
	Robot	:	Meca500;	
	Sent		:	BOOL;
	Buffered	:	BOOL;
END_VAR
VAR_OUTPUT
	Error		:	BOOL;
END_VAR
VAR
	Output_Params	:	ARRAY[1..6] OF REAL;
	FirstScan		:	BOOL;
END_VAR

        (*Collect Inputs and store them locally*)
Output_Params[1]:=Velocity_Limit;
Output_Params[2]:=0;
Output_Params[3]:=0;
Output_Params[4]:=0;
Output_Params[5]:=0;
Output_Params[6]:=0;


(* If Values have change, Reinitialise Outputs*)

IF FirstScan=0 OR Robot.Outputs.MotionCommand.Argument0 <> Output_Params[1] OR Robot.Outputs.MotionCommand.Argument1 <> Output_Params[2] OR Robot.Outputs.MotionCommand.Argument2 <> Output_Params[3] OR Robot.Outputs.MotionCommand.Argument3 <> Output_Params[4] OR Robot.Outputs.MotionCommand.Argument4 <> Output_Params[5] OR Robot.Outputs.MotionCommand.Argument5 <> Output_Params[6] THEN
	Buffered := FALSE;
	Sent := FALSE;
END_IF;

(*if not in legacy mode, Act Setpoint*)
IF Robot.Outputs.MoveID <> 0 THEN
    Robot.Outputs.MotionControl.SetPoint := TRUE;
END_IF;

(* To send _Move, send _Move ID *)
IF NOT Buffered AND NOT Sent THEN
    
    Robot.Outputs.MotionCommand.MoveCommand := Meca500_MotionCommandID.SET_CART_ANG_VEL;
    Robot.Outputs.MotionCommand.Argument0 := Output_Params[1];
	Robot.Outputs.MotionCommand.Argument1 := Output_Params[2];
	Robot.Outputs.MotionCommand.Argument2 := Output_Params[3];
	Robot.Outputs.MotionCommand.Argument3 := Output_Params[4];
	Robot.Outputs.MotionCommand.Argument4 := Output_Params[5];
	Robot.Outputs.MotionCommand.Argument5 := Output_Params[6];
    
    IF ExternalStateControl THEN
        IF ExternalMoveID <> 0 AND ExternalMoveID <> 32100 AND ExternalMoveID <> 32101 THEN
            Robot.Outputs.MoveID := ExternalMoveID;
            Sent := TRUE;
        END_IF;
        
    ELSE (*Not External Control*)
        IF Robot.Outputs.MoveID = 32100 THEN
            Robot.Outputs.MoveID := 32101;
        ELSIF Robot.Outputs.MoveID = 32101 THEN
            Robot.Outputs.MoveID := 32100;
        ELSIF Robot.Outputs.MoveID <> 32100 OR Robot.Outputs.MoveID <> 32101 THEN
            Robot.Outputs.MoveID := 32100;
        END_IF;
        Sent := TRUE;
    END_IF;
END_IF;

(* Check if _Move has been sent, if so, check if it was received *)
IF Sent THEN
    IF Robot.Outputs.MotionCommand.MoveCommand = Meca500_MotionCommandID.SET_CART_ANG_VEL THEN
        IF Robot.Outputs.MotionCommand.Argument0 = Output_Params[1] AND Robot.Outputs.MotionCommand.Argument1 = Output_Params[2] AND Robot.Outputs.MotionCommand.Argument2 = Output_Params[3] AND Robot.Outputs.MotionCommand.Argument3 = Output_Params[4] AND Robot.Outputs.MotionCommand.Argument4 = Output_Params[5] AND Robot.Outputs.MotionCommand.Argument5 = Output_Params[6] THEN
            IF Robot.Inputs.Motion.MoveID = Robot.Outputs.MoveID THEN
                Buffered := TRUE;
            END_IF;
        END_IF;
    END_IF;
END_IF;

(*If External _Move ID is equal to Internal, raise an error*)
IF ExternalMoveID = 32100 OR ExternalMoveID = 32101 THEN
    Error := TRUE;
END_IF;
FirstScan:=TRUE;

END_FUNCTION_BLOCK

// Device/Application/F1000_FBs/Meca500/SetConf
FUNCTION_BLOCK SetConf
VAR_INPUT
	Shoulder				:	REAL;
	Elbow					:	REAL;
	Wrist					:	REAL;
	ExternalStatecontrol 	:	BOOL;
	ExternalMoveID			:	UINT;
END_VAR
VAR_IN_OUT
	Robot	:	Meca500;	
	Sent		:	BOOL;
	Buffered	:	BOOL;
END_VAR
VAR_OUTPUT
	Error		:	BOOL;
END_VAR
VAR
	Output_Params	:	ARRAY[1..6] OF REAL;
	FirstScan		:	BOOL;
END_VAR

        (*Collect Inputs and store them locally*)
Output_Params[1]:=Shoulder;
Output_Params[2]:=Elbow;
Output_Params[3]:=Wrist;
Output_Params[4]:=0;
Output_Params[5]:=0;
Output_Params[6]:=0;


(* If Values have change, Reinitialise Outputs*)

IF FirstScan=0 OR Robot.Outputs.MotionCommand.Argument0 <> Output_Params[1] OR Robot.Outputs.MotionCommand.Argument1 <> Output_Params[2] OR Robot.Outputs.MotionCommand.Argument2 <> Output_Params[3] OR Robot.Outputs.MotionCommand.Argument3 <> Output_Params[4] OR Robot.Outputs.MotionCommand.Argument4 <> Output_Params[5] OR Robot.Outputs.MotionCommand.Argument5 <> Output_Params[6] THEN
	Buffered := FALSE;
	Sent := FALSE;
END_IF;


(*if not in legacy mode, Act Setpoint*)
IF Robot.Outputs.MoveID <> 0 THEN
    Robot.Outputs.MotionControl.SetPoint := TRUE;
END_IF;

(* To send _Move, send _Move ID *)
IF NOT Buffered AND NOT Sent THEN
    
    Robot.Outputs.MotionCommand.MoveCommand := Meca500_MotionCommandID.SET_CONF;
    Robot.Outputs.MotionCommand.Argument0 := Output_Params[1];
	Robot.Outputs.MotionCommand.Argument1 := Output_Params[2];
	Robot.Outputs.MotionCommand.Argument2 := Output_Params[3];
	Robot.Outputs.MotionCommand.Argument3 := Output_Params[4];
	Robot.Outputs.MotionCommand.Argument4 := Output_Params[5];
	Robot.Outputs.MotionCommand.Argument5 := Output_Params[6];
    
    IF ExternalStateControl THEN
        IF ExternalMoveID <> 0 AND ExternalMoveID <> 32150 AND ExternalMoveID <> 32151 THEN
            Robot.Outputs.MoveID := ExternalMoveID;
            Sent := TRUE;
        END_IF;
        
    ELSE (*Not External Control*)
        IF Robot.Outputs.MoveID = 32150 THEN
            Robot.Outputs.MoveID := 32151;
        ELSIF Robot.Outputs.MoveID = 32151 THEN
            Robot.Outputs.MoveID := 32150;
        ELSIF Robot.Outputs.MoveID <> 32150 OR Robot.Outputs.MoveID <> 32151 THEN
            Robot.Outputs.MoveID := 32150;
        END_IF;
        Sent := TRUE;
    END_IF;
END_IF;

(* Check if _Move has been sent, if so, check if it was received *)
IF Sent THEN
    IF Robot.Outputs.MotionCommand.MoveCommand = Meca500_MotionCommandID.SET_CONF THEN
        IF Robot.Outputs.MotionCommand.Argument0 = Output_Params[1] AND Robot.Outputs.MotionCommand.Argument1 = Output_Params[2] AND Robot.Outputs.MotionCommand.Argument2 = Output_Params[3] AND Robot.Outputs.MotionCommand.Argument3 = Output_Params[4] AND Robot.Outputs.MotionCommand.Argument4 = Output_Params[5] AND Robot.Outputs.MotionCommand.Argument5 = Output_Params[6] THEN
            IF Robot.Inputs.Motion.MoveID = Robot.Outputs.MoveID THEN
                Buffered := TRUE;
            END_IF;
        END_IF;
    END_IF;
END_IF;

(*If External _Move ID is equal to Internal, raise an error*)
IF ExternalMoveID = 32150 OR ExternalMoveID = 32151 THEN
    Error := TRUE;
END_IF;
FirstScan:=TRUE;

END_FUNCTION_BLOCK

// Device/Application/F1000_FBs/Meca500/SetConfTurn
FUNCTION_BLOCK SetConfTurn
VAR_INPUT
	Config					:	REAL;
	ExternalStatecontrol 	:	BOOL;
	ExternalMoveID			:	UINT;
END_VAR
VAR_IN_OUT
	Robot	:	Meca500;	
	Sent		:	BOOL;
	Buffered	:	BOOL;
END_VAR
VAR_OUTPUT
	Error		:	BOOL;
END_VAR
VAR
	Output_Params	:	ARRAY[1..6] OF REAL;
	FirstScan		:	Bool;
END_VAR

        (*Collect Inputs and store them locally*)
Output_Params[1]:=Config;
Output_Params[2]:=0;
Output_Params[3]:=0;
Output_Params[4]:=0;
Output_Params[5]:=0;
Output_Params[6]:=0;


(* If Values have change, Reinitialise Outputs*)

IF FirstScan=0 OR Robot.Outputs.MotionCommand.Argument0 <> Output_Params[1] OR Robot.Outputs.MotionCommand.Argument1 <> Output_Params[2] OR Robot.Outputs.MotionCommand.Argument2 <> Output_Params[3] OR Robot.Outputs.MotionCommand.Argument3 <> Output_Params[4] OR Robot.Outputs.MotionCommand.Argument4 <> Output_Params[5] OR Robot.Outputs.MotionCommand.Argument5 <> Output_Params[6] THEN
	Buffered := FALSE;
	Sent := FALSE;
END_IF;

(*if not in legacy mode, Act Setpoint*)
IF Robot.Outputs.MoveID <> 0 THEN
    Robot.Outputs.MotionControl.SetPoint := TRUE;
END_IF;

(* To send _Move, send _Move ID *)
IF NOT Buffered AND NOT Sent THEN
    
    Robot.Outputs.MotionCommand.MoveCommand := Meca500_MotionCommandID.SET_CONF_TURN;
    Robot.Outputs.MotionCommand.Argument0 := Output_Params[1];
	Robot.Outputs.MotionCommand.Argument1 := Output_Params[2];
	Robot.Outputs.MotionCommand.Argument2 := Output_Params[3];
	Robot.Outputs.MotionCommand.Argument3 := Output_Params[4];
	Robot.Outputs.MotionCommand.Argument4 := Output_Params[5];
	Robot.Outputs.MotionCommand.Argument5 := Output_Params[6];
    
    IF ExternalStateControl THEN
        IF ExternalMoveID <> 0 AND ExternalMoveID <> 32250 AND ExternalMoveID <> 32251 THEN
            Robot.Outputs.MoveID := ExternalMoveID;
            Sent := TRUE;
        END_IF;
        
    ELSE (*Not External Control*)
        IF Robot.Outputs.MoveID = 32250 THEN
            Robot.Outputs.MoveID := 32251;
        ELSIF Robot.Outputs.MoveID = 32251 THEN
            Robot.Outputs.MoveID := 32250;
        ELSIF Robot.Outputs.MoveID <> 32250 OR Robot.Outputs.MoveID <> 32251 THEN
            Robot.Outputs.MoveID := 32250;
        END_IF;
        Sent := TRUE;
    END_IF;
END_IF;

(* Check if _Move has been sent, if so, check if it was received *)
IF Sent THEN
    IF Robot.Outputs.MotionCommand.MoveCommand = Meca500_MotionCommandID.SET_CONF_TURN THEN
        IF Robot.Outputs.MotionCommand.Argument0 = Output_Params[1] AND Robot.Outputs.MotionCommand.Argument1 = Output_Params[2] AND Robot.Outputs.MotionCommand.Argument2 = Output_Params[3] AND Robot.Outputs.MotionCommand.Argument3 = Output_Params[4] AND Robot.Outputs.MotionCommand.Argument4 = Output_Params[5] AND Robot.Outputs.MotionCommand.Argument5 = Output_Params[6] THEN
            IF Robot.Inputs.Motion.MoveID = Robot.Outputs.MoveID THEN
                Buffered := TRUE;
            END_IF;
        END_IF;
    END_IF;
END_IF;

(*If External _Move ID is equal to Internal, raise an error*)
IF ExternalMoveID = 32250 OR ExternalMoveID = 32251 THEN
    Error := TRUE;
END_IF;
FirstScan:=TRUE;

END_FUNCTION_BLOCK

// Device/Application/F1000_FBs/Meca500/SetGripperForce
FUNCTION_BLOCK SetGripperForce
VAR_INPUT
	Force					:	REAL;
	ExternalStatecontrol 	:	BOOL;
	ExternalMoveID			:	UINT;
END_VAR
VAR_IN_OUT
	Robot	:	Meca500;	
	Sent		:	BOOL;
	Buffered	:	BOOL;
END_VAR
VAR_OUTPUT
	Error		:	BOOL;
END_VAR
VAR
	Output_Params	:	ARRAY[1..6] OF REAL;
	FirstScan		:	BOOL;
END_VAR

        (*Collect Inputs and store them locally*)
Output_Params[1]:=Force;
Output_Params[2]:=0;
Output_Params[3]:=0;
Output_Params[4]:=0;
Output_Params[5]:=0;
Output_Params[6]:=0;


(* If Values have change, Reinitialise Outputs*)

IF FirstScan=0 OR Robot.Outputs.MotionCommand.Argument0 <> Output_Params[1] OR Robot.Outputs.MotionCommand.Argument1 <> Output_Params[2] OR Robot.Outputs.MotionCommand.Argument2 <> Output_Params[3] OR Robot.Outputs.MotionCommand.Argument3 <> Output_Params[4] OR Robot.Outputs.MotionCommand.Argument4 <> Output_Params[5] OR Robot.Outputs.MotionCommand.Argument5 <> Output_Params[6] THEN
	Buffered := FALSE;
	Sent := FALSE;
END_IF;


(*if not in legacy mode, Act Setpoint*)
IF Robot.Outputs.MoveID <> 0 THEN
    Robot.Outputs.MotionControl.SetPoint := TRUE;
END_IF;

(* To send _Move, send _Move ID *)
IF NOT Buffered AND NOT Sent THEN
    
    Robot.Outputs.MotionCommand.MoveCommand := Meca500_MotionCommandID.SET_GRIPPER_FORCE;
    Robot.Outputs.MotionCommand.Argument0 := Output_Params[1];
	Robot.Outputs.MotionCommand.Argument1 := Output_Params[2];
	Robot.Outputs.MotionCommand.Argument2 := Output_Params[3];
	Robot.Outputs.MotionCommand.Argument3 := Output_Params[4];
	Robot.Outputs.MotionCommand.Argument4 := Output_Params[5];
	Robot.Outputs.MotionCommand.Argument5 := Output_Params[6];
    
    IF ExternalStateControl THEN
        IF ExternalMoveID <> 0 AND ExternalMoveID <> 32200 AND ExternalMoveID <> 32201 THEN
            Robot.Outputs.MoveID := ExternalMoveID;
            Sent := TRUE;
        END_IF;
        
    ELSE (*Not External Control*)
        IF Robot.Outputs.MoveID = 32200 THEN
            Robot.Outputs.MoveID := 32201;
        ELSIF Robot.Outputs.MoveID = 32201 THEN
            Robot.Outputs.MoveID := 32200;
        ELSIF Robot.Outputs.MoveID <> 32200 OR Robot.Outputs.MoveID <> 32201 THEN
            Robot.Outputs.MoveID := 32200;
        END_IF;
        Sent := TRUE;
    END_IF;
END_IF;

(* Check if _Move has been sent, if so, check if it was received *)
IF Sent THEN
    IF Robot.Outputs.MotionCommand.MoveCommand = Meca500_MotionCommandID.SET_GRIPPER_FORCE THEN
        IF Robot.Outputs.MotionCommand.Argument0 = Output_Params[1] AND Robot.Outputs.MotionCommand.Argument1 = Output_Params[2] AND Robot.Outputs.MotionCommand.Argument2 = Output_Params[3] AND Robot.Outputs.MotionCommand.Argument3 = Output_Params[4] AND Robot.Outputs.MotionCommand.Argument4 = Output_Params[5] AND Robot.Outputs.MotionCommand.Argument5 = Output_Params[6] THEN
            IF Robot.Inputs.Motion.MoveID = Robot.Outputs.MoveID THEN
                Buffered := TRUE;
            END_IF;
        END_IF;
    END_IF;
END_IF;

(*If External _Move ID is equal to Internal, raise an error*)
IF ExternalMoveID = 32200 OR ExternalMoveID = 32201 THEN
    Error := TRUE;
END_IF;
FirstScan:=TRUE;

END_FUNCTION_BLOCK

// Device/Application/F1000_FBs/Meca500/SetGripperRange
FUNCTION_BLOCK SetGripperRange
VAR_INPUT
	Minimum					:	REAL;
	Maximum					:	REAL;
	ExternalStatecontrol 	:	BOOL;
	ExternalMoveID			:	UINT;
END_VAR
VAR_IN_OUT
	Robot	:	Meca500;	
	Sent		:	BOOL;
	Buffered	:	BOOL;
END_VAR
VAR_OUTPUT
	Error		:	BOOL;
END_VAR
VAR
	Output_Params	:	ARRAY[1..6] OF REAL;
	FirstScan		:	BOOL;
END_VAR

        (*Collect Inputs and store them locally*)
Output_Params[1]:=Minimum;
Output_Params[2]:=Maximum;
Output_Params[3]:=0;
Output_Params[4]:=0;
Output_Params[5]:=0;
Output_Params[6]:=0;


(* If Values have change, Reinitialise Outputs*)

IF FirstScan=0 OR Robot.Outputs.MotionCommand.Argument0 <> Output_Params[1] OR Robot.Outputs.MotionCommand.Argument1 <> Output_Params[2] OR Robot.Outputs.MotionCommand.Argument2 <> Output_Params[3] OR Robot.Outputs.MotionCommand.Argument3 <> Output_Params[4] OR Robot.Outputs.MotionCommand.Argument4 <> Output_Params[5] OR Robot.Outputs.MotionCommand.Argument5 <> Output_Params[6] THEN
	Buffered := FALSE;
	Sent := FALSE;
END_IF;

(*if not in legacy mode, Act Setpoint*)
IF Robot.Outputs.MoveID <> 0 THEN
    Robot.Outputs.MotionControl.SetPoint := TRUE;
END_IF;

(* To send _Move, send _Move ID *)
IF NOT Buffered AND NOT Sent THEN
    
    Robot.Outputs.MotionCommand.MoveCommand := Meca500_MotionCommandID.SET_GRIPPER_RANGE;
    Robot.Outputs.MotionCommand.Argument0 := Output_Params[1];
	Robot.Outputs.MotionCommand.Argument1 := Output_Params[2];
	Robot.Outputs.MotionCommand.Argument2 := Output_Params[3];
	Robot.Outputs.MotionCommand.Argument3 := Output_Params[4];
	Robot.Outputs.MotionCommand.Argument4 := Output_Params[5];
	Robot.Outputs.MotionCommand.Argument5 := Output_Params[6];
    
    IF ExternalStateControl THEN
        IF ExternalMoveID <> 0 AND ExternalMoveID <> 32310 AND ExternalMoveID <> 32311 THEN
            Robot.Outputs.MoveID := ExternalMoveID;
            Sent := TRUE;
        END_IF;
        
    ELSE (*Not External Control*)
        IF Robot.Outputs.MoveID = 32310 THEN
            Robot.Outputs.MoveID := 32311;
        ELSIF Robot.Outputs.MoveID = 32311 THEN
            Robot.Outputs.MoveID := 32310;
        ELSIF Robot.Outputs.MoveID <> 32310 OR Robot.Outputs.MoveID <> 32311 THEN
            Robot.Outputs.MoveID := 32310;
        END_IF;
        Sent := TRUE;
    END_IF;
END_IF;

(* Check if _Move has been sent, if so, check if it was received *)
IF Sent THEN
    IF Robot.Outputs.MotionCommand.MoveCommand = Meca500_MotionCommandID.SET_GRIPPER_RANGE THEN
        IF Robot.Outputs.MotionCommand.Argument0 = Output_Params[1] AND Robot.Outputs.MotionCommand.Argument1 = Output_Params[2] AND Robot.Outputs.MotionCommand.Argument2 = Output_Params[3] AND Robot.Outputs.MotionCommand.Argument3 = Output_Params[4] AND Robot.Outputs.MotionCommand.Argument4 = Output_Params[5] AND Robot.Outputs.MotionCommand.Argument5 = Output_Params[6] THEN
            IF Robot.Inputs.Motion.MoveID = Robot.Outputs.MoveID THEN
                Buffered := TRUE;
            END_IF;
        END_IF;
    END_IF;
END_IF;

(*If External _Move ID is equal to Internal, raise an error*)
IF ExternalMoveID = 32310 OR ExternalMoveID = 32311 THEN
    Error := TRUE;
END_IF;
FirstScan:=TRUE;

END_FUNCTION_BLOCK

// Device/Application/F1000_FBs/Meca500/SetGripperVel
FUNCTION_BLOCK SetGripperVel
VAR_INPUT
	Speed					:	REAL;
	ExternalStatecontrol 	:	BOOL;
	ExternalMoveID			:	UINT;
END_VAR
VAR_IN_OUT
	Robot	:	Meca500;	
	Sent		:	BOOL;
	Buffered	:	BOOL;
END_VAR
VAR_OUTPUT
	Error		:	BOOL;
END_VAR
VAR
	Output_Params	:	ARRAY[1..6] OF REAL;
	FirstScan		:	BOOL;
END_VAR

        (*Collect Inputs and store them locally*)
Output_Params[1]:=Speed;
Output_Params[2]:=0;
Output_Params[3]:=0;
Output_Params[4]:=0;
Output_Params[5]:=0;
Output_Params[6]:=0;


(* If Values have change, Reinitialise Outputs*)

IF FirstScan=0 OR Robot.Outputs.MotionCommand.Argument0 <> Output_Params[1] OR Robot.Outputs.MotionCommand.Argument1 <> Output_Params[2] OR Robot.Outputs.MotionCommand.Argument2 <> Output_Params[3] OR Robot.Outputs.MotionCommand.Argument3 <> Output_Params[4] OR Robot.Outputs.MotionCommand.Argument4 <> Output_Params[5] OR Robot.Outputs.MotionCommand.Argument5 <> Output_Params[6] THEN
	Buffered := FALSE;
	Sent := FALSE;
END_IF;

(*if not in legacy mode, Act Setpoint*)
IF Robot.Outputs.MoveID <> 0 THEN
    Robot.Outputs.MotionControl.SetPoint := TRUE;
END_IF;

(* To send _Move, send _Move ID *)
IF NOT Buffered AND NOT Sent THEN
    
    Robot.Outputs.MotionCommand.MoveCommand := Meca500_MotionCommandID.SET_GRIPPER_VEL;
    Robot.Outputs.MotionCommand.Argument0 := Output_Params[1];
	Robot.Outputs.MotionCommand.Argument1 := Output_Params[2];
	Robot.Outputs.MotionCommand.Argument2 := Output_Params[3];
	Robot.Outputs.MotionCommand.Argument3 := Output_Params[4];
	Robot.Outputs.MotionCommand.Argument4 := Output_Params[5];
	Robot.Outputs.MotionCommand.Argument5 := Output_Params[6];
    
    IF ExternalStateControl THEN
        IF ExternalMoveID <> 0 AND ExternalMoveID <> 32190 AND ExternalMoveID <> 32191 THEN
            Robot.Outputs.MoveID := ExternalMoveID;
            Sent := TRUE;
        END_IF;
        
    ELSE (*Not External Control*)
        IF Robot.Outputs.MoveID = 32190 THEN
            Robot.Outputs.MoveID := 32191;
        ELSIF Robot.Outputs.MoveID = 32191 THEN
            Robot.Outputs.MoveID := 32190;
        ELSIF Robot.Outputs.MoveID <> 32190 OR Robot.Outputs.MoveID <> 32191 THEN
            Robot.Outputs.MoveID := 32190;
        END_IF;
        Sent := TRUE;
    END_IF;
END_IF;

(* Check if _Move has been sent, if so, check if it was received *)
IF Sent THEN
    IF Robot.Outputs.MotionCommand.MoveCommand = Meca500_MotionCommandID.SET_GRIPPER_VEL THEN
        IF Robot.Outputs.MotionCommand.Argument0 = Output_Params[1] AND Robot.Outputs.MotionCommand.Argument1 = Output_Params[2] AND Robot.Outputs.MotionCommand.Argument2 = Output_Params[3] AND Robot.Outputs.MotionCommand.Argument3 = Output_Params[4] AND Robot.Outputs.MotionCommand.Argument4 = Output_Params[5] AND Robot.Outputs.MotionCommand.Argument5 = Output_Params[6] THEN
            IF Robot.Inputs.Motion.MoveID = Robot.Outputs.MoveID THEN
                Buffered := TRUE;
            END_IF;
        END_IF;
    END_IF;
END_IF;

(*If External _Move ID is equal to Internal, raise an error*)
IF ExternalMoveID = 32190 OR ExternalMoveID = 32191 THEN
    Error := TRUE;
END_IF;
FirstScan:=TRUE;

END_FUNCTION_BLOCK

// Device/Application/F1000_FBs/Meca500/SetJointAcc
FUNCTION_BLOCK SetJointAcc
VAR_INPUT
	Acceleration_Percentage			:	REAL;
	ExternalStatecontrol 	:	BOOL;
	ExternalMoveID			:	UINT;
END_VAR
VAR_IN_OUT
	Robot	:	Meca500;	
	Sent		:	BOOL;
	Buffered	:	BOOL;
END_VAR
VAR_OUTPUT
	Error		:	BOOL;
END_VAR
VAR
	Output_Params	:	ARRAY[1..6] OF REAL;
	FirstScan		:	Bool;
END_VAR

        (*Collect Inputs and store them locally*)
Output_Params[1]:= Acceleration_Percentage;
Output_Params[2]:=0;
Output_Params[3]:=0;
Output_Params[4]:=0;
Output_Params[5]:=0;
Output_Params[6]:=0;


(* If Values have change, Reinitialise Outputs*)

IF FirstScan=0 OR Robot.Outputs.MotionCommand.Argument0 <> Output_Params[1] OR Robot.Outputs.MotionCommand.Argument1 <> Output_Params[2] OR Robot.Outputs.MotionCommand.Argument2 <> Output_Params[3] OR Robot.Outputs.MotionCommand.Argument3 <> Output_Params[4] OR Robot.Outputs.MotionCommand.Argument4 <> Output_Params[5] OR Robot.Outputs.MotionCommand.Argument5 <> Output_Params[6] THEN
	Buffered := FALSE;
	Sent := FALSE;
END_IF;

(*if not in legacy mode, Act Setpoint*)
IF Robot.Outputs.MoveID <> 0 THEN
    Robot.Outputs.MotionControl.SetPoint := TRUE;
END_IF;

(* To send _Move, send _Move ID *)
IF NOT Buffered AND NOT Sent THEN
    
    Robot.Outputs.MotionCommand.MoveCommand := Meca500_MotionCommandID.SET_JOINT_ACC;
    Robot.Outputs.MotionCommand.Argument0 := Output_Params[1];
	Robot.Outputs.MotionCommand.Argument1 := Output_Params[2];
	Robot.Outputs.MotionCommand.Argument2 := Output_Params[3];
	Robot.Outputs.MotionCommand.Argument3 := Output_Params[4];
	Robot.Outputs.MotionCommand.Argument4 := Output_Params[5];
	Robot.Outputs.MotionCommand.Argument5 := Output_Params[6];
    
    IF ExternalStateControl THEN
        IF ExternalMoveID <> 0 AND ExternalMoveID <> 32090 AND ExternalMoveID <> 32091 THEN
            Robot.Outputs.MoveID := ExternalMoveID;
            Sent := TRUE;
        END_IF;
        
    ELSE (*Not External Control*)
        IF Robot.Outputs.MoveID = 32090 THEN
            Robot.Outputs.MoveID := 32091;
        ELSIF Robot.Outputs.MoveID = 32091 THEN
            Robot.Outputs.MoveID := 32090;
        ELSIF Robot.Outputs.MoveID <> 32090 OR Robot.Outputs.MoveID <> 32091 THEN
            Robot.Outputs.MoveID := 32090;
        END_IF;
        Sent := TRUE;
    END_IF;
END_IF;

(* Check if _Move has been sent, if so, check if it was received *)
IF Sent THEN
    IF Robot.Outputs.MotionCommand.MoveCommand = Meca500_MotionCommandID.SET_JOINT_ACC THEN
        IF Robot.Outputs.MotionCommand.Argument0 = Output_Params[1] AND Robot.Outputs.MotionCommand.Argument1 = Output_Params[2] AND Robot.Outputs.MotionCommand.Argument2 = Output_Params[3] AND Robot.Outputs.MotionCommand.Argument3 = Output_Params[4] AND Robot.Outputs.MotionCommand.Argument4 = Output_Params[5] AND Robot.Outputs.MotionCommand.Argument5 = Output_Params[6] THEN
            IF Robot.Inputs.Motion.MoveID = Robot.Outputs.MoveID THEN
                Buffered := TRUE;
            END_IF;
        END_IF;
    END_IF;
END_IF;

(*If External _Move ID is equal to Internal, raise an error*)
IF ExternalMoveID = 32090 OR ExternalMoveID = 32091 THEN
    Error := TRUE;
END_IF;
FirstScan:=TRUE;

END_FUNCTION_BLOCK

// Device/Application/F1000_FBs/Meca500/SetJointsVelLimit
FUNCTION_BLOCK SetJointsVelLimit

VAR_INPUT
	Velocity_Limit_Percentage					:	REAL;
	ExternalStatecontrol 	:	BOOL;
	ExternalMoveID			:	UINT;
END_VAR

VAR_IN_OUT
	Robot	:	Meca500;	
	Sent		:	BOOL;
	Buffered	:	BOOL;
END_VAR

VAR_OUTPUT
	Error		:	BOOL;
END_VAR

VAR
	Output_Params	:	ARRAY[1..6] OF REAL;
	FirstScan		:	Bool;
END_VAR

       (*Collect Inputs and store them locally*)
Output_Params[1]:=Velocity_Limit_Percentage;
Output_Params[2]:=0;
Output_Params[3]:=0;
Output_Params[4]:=0;
Output_Params[5]:=0;
Output_Params[6]:=0;

(* If Values have change, Reinitialise Outputs*)

IF FirstScan=0 OR Robot.Outputs.MotionCommand.Argument0 <> Output_Params[1] OR Robot.Outputs.MotionCommand.Argument1 <> Output_Params[2] OR Robot.Outputs.MotionCommand.Argument2 <> Output_Params[3] OR Robot.Outputs.MotionCommand.Argument3 <> Output_Params[4] OR Robot.Outputs.MotionCommand.Argument4 <> Output_Params[5] OR Robot.Outputs.MotionCommand.Argument5 <> Output_Params[6] THEN
	Buffered := FALSE;
	Sent := FALSE;
END_IF;

(*if not in legacy mode, Act Setpoint*)
IF Robot.Outputs.MoveID <> 0 THEN
    Robot.Outputs.MotionControl.SetPoint := TRUE;
END_IF;

(* To send _Move, send _Move ID *)
IF NOT Buffered AND NOT Sent THEN
    
    Robot.Outputs.MotionCommand.MoveCommand := Meca500_MotionCommandID.SET_JOINT_VEL_LIMIT;
    Robot.Outputs.MotionCommand.Argument0 := Output_Params[1];
	Robot.Outputs.MotionCommand.Argument1 := Output_Params[2];
	Robot.Outputs.MotionCommand.Argument2 := Output_Params[3];
	Robot.Outputs.MotionCommand.Argument3 := Output_Params[4];
	Robot.Outputs.MotionCommand.Argument4 := Output_Params[5];
	Robot.Outputs.MotionCommand.Argument5 := Output_Params[6];
    
    IF ExternalStateControl THEN
        IF ExternalMoveID <> 0 AND ExternalMoveID <> 32330 AND ExternalMoveID <> 32331 THEN
            Robot.Outputs.MoveID := ExternalMoveID;
            Sent := TRUE;
        END_IF;
        
    ELSE (*Not External Control*)
        IF Robot.Outputs.MoveID = 32330 THEN
            Robot.Outputs.MoveID :=32331;
        ELSIF Robot.Outputs.MoveID = 32331 THEN
            Robot.Outputs.MoveID := 32330;
        ELSIF Robot.Outputs.MoveID <> 32330 OR Robot.Outputs.MoveID <> 32331 THEN
            Robot.Outputs.MoveID := 32330;
        END_IF;
        Sent := TRUE;
    END_IF;
END_IF;

(* Check if _Move has been sent, if so, check if it was received *)
IF Sent THEN
    IF Robot.Outputs.MotionCommand.MoveCommand = Meca500_MotionCommandID.SET_JOINT_VEL_LIMIT THEN
        IF Robot.Outputs.MotionCommand.Argument0 = Output_Params[1] AND Robot.Outputs.MotionCommand.Argument1 = Output_Params[2] AND Robot.Outputs.MotionCommand.Argument2 = Output_Params[3] AND Robot.Outputs.MotionCommand.Argument3 = Output_Params[4] AND Robot.Outputs.MotionCommand.Argument4 = Output_Params[5] AND Robot.Outputs.MotionCommand.Argument5 = Output_Params[6] THEN
            IF Robot.Inputs.Motion.MoveID = Robot.Outputs.MoveID THEN
                Buffered := TRUE;
            END_IF;
        END_IF;
    END_IF;
END_IF;

(*If External _Move ID is equal to Internal, raise an error*)
IF ExternalMoveID = 32330 OR ExternalMoveID = 32331 THEN
    Error := TRUE;
END_IF;
FirstScan:=TRUE;

END_FUNCTION_BLOCK

// Device/Application/F1000_FBs/Meca500/SetTorqueLimitCfg
FUNCTION_BLOCK SetTorqueLimitCfg
VAR_INPUT
	Severity				:	REAL;
	Mode					:	REAL;
	ExternalStatecontrol 	:	BOOL;
	ExternalMoveID			:	UINT;
END_VAR
VAR_IN_OUT
	Robot	:	Meca500;	
	Sent		:	BOOL;
	Buffered	:	BOOL;
END_VAR
VAR_OUTPUT
	Error		:	BOOL;
END_VAR
VAR
	Output_Params	:	ARRAY[1..6] OF REAL;
	FirstScan		:	Bool;
END_VAR

        (*Collect Inputs and store them locally*)
Output_Params[1]:=Severity;
Output_Params[2]:=Mode;
Output_Params[3]:=0;
Output_Params[4]:=0;
Output_Params[5]:=0;
Output_Params[6]:=0;


(* If Values have change, Reinitialise Outputs*)

IF FirstScan=0 OR Robot.Outputs.MotionCommand.Argument0 <> Output_Params[1] OR Robot.Outputs.MotionCommand.Argument1 <> Output_Params[2] OR Robot.Outputs.MotionCommand.Argument2 <> Output_Params[3] OR Robot.Outputs.MotionCommand.Argument3 <> Output_Params[4] OR Robot.Outputs.MotionCommand.Argument4 <> Output_Params[5] OR Robot.Outputs.MotionCommand.Argument5 <> Output_Params[6] THEN
	Buffered := FALSE;
	Sent := FALSE;
END_IF;

(*if not in legacy mode, Act Setpoint*)
IF Robot.Outputs.MoveID <> 0 THEN
    Robot.Outputs.MotionControl.SetPoint := TRUE;
END_IF;

(* To send _Move, send _Move ID *)
IF NOT Buffered AND NOT Sent THEN
    
    Robot.Outputs.MotionCommand.MoveCommand := Meca500_MotionCommandID.SET_TORQUE_LIMIT_CFG;
    Robot.Outputs.MotionCommand.Argument0 := Output_Params[1];
	Robot.Outputs.MotionCommand.Argument1 := Output_Params[2];
	Robot.Outputs.MotionCommand.Argument2 := Output_Params[3];
	Robot.Outputs.MotionCommand.Argument3 := Output_Params[4];
	Robot.Outputs.MotionCommand.Argument4 := Output_Params[5];
	Robot.Outputs.MotionCommand.Argument5 := Output_Params[6];
    
    IF ExternalStateControl THEN
        IF ExternalMoveID <> 0 AND ExternalMoveID <> 32280 AND ExternalMoveID <> 32281 THEN
            Robot.Outputs.MoveID := ExternalMoveID;
            Sent := TRUE;
        END_IF;
        
    ELSE (*Not External Control*)
        IF Robot.Outputs.MoveID = 32280 THEN
            Robot.Outputs.MoveID := 32281;
        ELSIF Robot.Outputs.MoveID = 32281 THEN
            Robot.Outputs.MoveID := 32280;
        ELSIF Robot.Outputs.MoveID <> 32280 OR Robot.Outputs.MoveID <> 32281 THEN
            Robot.Outputs.MoveID := 32280;
        END_IF;
        Sent := TRUE;
    END_IF;
END_IF;

(* Check if _Move has been sent, if so, check if it was received *)
IF Sent THEN
    IF Robot.Outputs.MotionCommand.MoveCommand = Meca500_MotionCommandID.SET_TORQUE_LIMIT_CFG THEN
        IF Robot.Outputs.MotionCommand.Argument0 = Output_Params[1] AND Robot.Outputs.MotionCommand.Argument1 = Output_Params[2] AND Robot.Outputs.MotionCommand.Argument2 = Output_Params[3] AND Robot.Outputs.MotionCommand.Argument3 = Output_Params[4] AND Robot.Outputs.MotionCommand.Argument4 = Output_Params[5] AND Robot.Outputs.MotionCommand.Argument5 = Output_Params[6] THEN
            IF Robot.Inputs.Motion.MoveID = Robot.Outputs.MoveID THEN
                Buffered := TRUE;
            END_IF;
        END_IF;
    END_IF;
END_IF;

(*If External _Move ID is equal to Internal, raise an error*)
IF ExternalMoveID = 32280 OR ExternalMoveID = 32281 THEN
    Error := TRUE;
END_IF;
FirstScan:=TRUE;

END_FUNCTION_BLOCK

// Device/Application/F1000_FBs/Meca500/SetTorqueLimits
FUNCTION_BLOCK SetTorqueLimits
VAR_INPUT
	Joints_Limit					:	ARRAY[1..6]OF REAL;
	ExternalStatecontrol 	:	BOOL;
	ExternalMoveID			:	UINT;
END_VAR
VAR_IN_OUT
	Robot	:	Meca500;	
	Sent		:	BOOL;
	Buffered	:	BOOL;
END_VAR
VAR_OUTPUT
	Error		:	BOOL;
END_VAR
VAR
	Output_Params	:	ARRAY[1..6] OF REAL;
	FirstScan		:	BOOL;
END_VAR

        (*Collect Inputs and store them locally*)
Output_Params[1]:=Joints_Limit[1];
Output_Params[2]:=Joints_Limit[2];
Output_Params[3]:=Joints_Limit[3];
Output_Params[4]:=Joints_Limit[4];
Output_Params[5]:=Joints_Limit[5];
Output_Params[6]:=Joints_Limit[6];


(* If Values have change, Reinitialise Outputs*)

IF FirstScan=0 OR Robot.Outputs.MotionCommand.Argument0 <> Output_Params[1] OR Robot.Outputs.MotionCommand.Argument1 <> Output_Params[2] OR Robot.Outputs.MotionCommand.Argument2 <> Output_Params[3] OR Robot.Outputs.MotionCommand.Argument3 <> Output_Params[4] OR Robot.Outputs.MotionCommand.Argument4 <> Output_Params[5] OR Robot.Outputs.MotionCommand.Argument5 <> Output_Params[6] THEN
	Buffered := FALSE;
	Sent := FALSE;
END_IF;

(*if not in legacy mode, Act Setpoint*)
IF Robot.Outputs.MoveID <> 0 THEN
    Robot.Outputs.MotionControl.SetPoint := TRUE;
END_IF;

(* To send _Move, send _Move ID *)
IF NOT Buffered AND NOT Sent THEN
    
    Robot.Outputs.MotionCommand.MoveCommand := Meca500_MotionCommandID.SET_TORQUE_LIMITS;
    Robot.Outputs.MotionCommand.Argument0 := Output_Params[1];
	Robot.Outputs.MotionCommand.Argument1 := Output_Params[2];
	Robot.Outputs.MotionCommand.Argument2 := Output_Params[3];
	Robot.Outputs.MotionCommand.Argument3 := Output_Params[4];
	Robot.Outputs.MotionCommand.Argument4 := Output_Params[5];
	Robot.Outputs.MotionCommand.Argument5 := Output_Params[6];
    
    IF ExternalStateControl THEN
        IF ExternalMoveID <> 0 AND ExternalMoveID <> 32270 AND ExternalMoveID <> 32271 THEN
            Robot.Outputs.MoveID := ExternalMoveID;
            Sent := TRUE;
        END_IF;
        
    ELSE (*Not External Control*)
        IF Robot.Outputs.MoveID = 32270 THEN
            Robot.Outputs.MoveID := 32271;
        ELSIF Robot.Outputs.MoveID = 32271 THEN
            Robot.Outputs.MoveID := 32270;
        ELSIF Robot.Outputs.MoveID <> 32270 OR Robot.Outputs.MoveID <> 32271 THEN
            Robot.Outputs.MoveID := 32270;
        END_IF;
        Sent := TRUE;
    END_IF;
END_IF;

(* Check if _Move has been sent, if so, check if it was received *)
IF Sent THEN
    IF Robot.Outputs.MotionCommand.MoveCommand = Meca500_MotionCommandID.SET_TORQUE_LIMITS THEN
        IF Robot.Outputs.MotionCommand.Argument0 = Output_Params[1] AND Robot.Outputs.MotionCommand.Argument1 = Output_Params[2] AND Robot.Outputs.MotionCommand.Argument2 = Output_Params[3] AND Robot.Outputs.MotionCommand.Argument3 = Output_Params[4] AND Robot.Outputs.MotionCommand.Argument4 = Output_Params[5] AND Robot.Outputs.MotionCommand.Argument5 = Output_Params[6] THEN
            IF Robot.Inputs.Motion.MoveID = Robot.Outputs.MoveID THEN
                Buffered := TRUE;
            END_IF;
        END_IF;
    END_IF;
END_IF;

(*If External _Move ID is equal to Internal, raise an error*)
IF ExternalMoveID = 32270 OR ExternalMoveID = 32271 THEN
    Error := TRUE;
END_IF;
FirstScan:=TRUE;

END_FUNCTION_BLOCK

// Device/Application/F1000_FBs/Meca500/SetValveState
FUNCTION_BLOCK SetValveState
VAR_INPUT
	V1					:	REAL;
	V2					:	REAL;
	ExternalStatecontrol 	:	BOOL;
	ExternalMoveID			:	UINT;
END_VAR
VAR_IN_OUT
	Robot	:	Meca500;	
	Sent		:	BOOL;
	Buffered	:	BOOL;
END_VAR
VAR_OUTPUT
	Error		:	BOOL;
END_VAR
VAR
	Output_Params	:	ARRAY[1..6] OF REAL;
	FirstScan		:	Bool;
END_VAR

        (*Collect Inputs and store them locally*)
Output_Params[1]:=V1;
Output_Params[2]:=V2;
Output_Params[3]:=0;
Output_Params[4]:=0;
Output_Params[5]:=0;
Output_Params[6]:=0;


(* If Values have change, Reinitialise Outputs*)

IF FirstScan=0 OR Robot.Outputs.MotionCommand.Argument0 <> Output_Params[1] OR Robot.Outputs.MotionCommand.Argument1 <> Output_Params[2] OR Robot.Outputs.MotionCommand.Argument2 <> Output_Params[3] OR Robot.Outputs.MotionCommand.Argument3 <> Output_Params[4] OR Robot.Outputs.MotionCommand.Argument4 <> Output_Params[5] OR Robot.Outputs.MotionCommand.Argument5 <> Output_Params[6] THEN
	Buffered := FALSE;
	Sent := FALSE;
END_IF;

(*if not in legacy mode, Act Setpoint*)
IF Robot.Outputs.MoveID <> 0 THEN
    Robot.Outputs.MotionControl.SetPoint := TRUE;
END_IF;

(* To send _Move, send _Move ID *)
IF NOT Buffered AND NOT Sent THEN
    
    Robot.Outputs.MotionCommand.MoveCommand := Meca500_MotionCommandID.SET_VALVE_STATE;
    Robot.Outputs.MotionCommand.Argument0 := Output_Params[1];
	Robot.Outputs.MotionCommand.Argument1 := Output_Params[2];
	Robot.Outputs.MotionCommand.Argument2 := Output_Params[3];
	Robot.Outputs.MotionCommand.Argument3 := Output_Params[4];
	Robot.Outputs.MotionCommand.Argument4 := Output_Params[5];
	Robot.Outputs.MotionCommand.Argument5 := Output_Params[6];
    
    IF ExternalStateControl THEN
        IF ExternalMoveID <> 0 AND ExternalMoveID <> 32300 AND ExternalMoveID <> 32301 THEN
            Robot.Outputs.MoveID := ExternalMoveID;
            Sent := TRUE;
        END_IF;
        
    ELSE (*Not External Control*)
        IF Robot.Outputs.MoveID = 32300 THEN
            Robot.Outputs.MoveID := 32301;
        ELSIF Robot.Outputs.MoveID = 32301 THEN
            Robot.Outputs.MoveID := 32300;
        ELSIF Robot.Outputs.MoveID <> 32300 OR Robot.Outputs.MoveID <> 32301 THEN
            Robot.Outputs.MoveID := 32300;
        END_IF;
        Sent := TRUE;
    END_IF;
END_IF;

(* Check if _Move has been sent, if so, check if it was received *)
IF Sent THEN
    IF Robot.Outputs.MotionCommand.MoveCommand = Meca500_MotionCommandID.SET_VALVE_STATE THEN
        IF Robot.Outputs.MotionCommand.Argument0 = Output_Params[1] AND Robot.Outputs.MotionCommand.Argument1 = Output_Params[2] AND Robot.Outputs.MotionCommand.Argument2 = Output_Params[3] AND Robot.Outputs.MotionCommand.Argument3 = Output_Params[4] AND Robot.Outputs.MotionCommand.Argument4 = Output_Params[5] AND Robot.Outputs.MotionCommand.Argument5 = Output_Params[6] THEN
            IF Robot.Inputs.Motion.MoveID = Robot.Outputs.MoveID THEN
                Buffered := TRUE;
            END_IF;
        END_IF;
    END_IF;
END_IF;

(*If External _Move ID is equal to Internal, raise an error*)
IF ExternalMoveID = 32300 OR ExternalMoveID = 32301 THEN
    Error := TRUE;
END_IF;
FirstScan:=TRUE;

END_FUNCTION_BLOCK

// Device/Application/F1000_FBs/Meca500/SetVelTimeout
FUNCTION_BLOCK SetVelTimeout
VAR_INPUT
	Seconds					:	REAL;
	ExternalStatecontrol 	:	BOOL;
	ExternalMoveID			:	UINT;
END_VAR
VAR_IN_OUT
	Robot	:	Meca500;	
	Sent		:	BOOL;
	Buffered	:	BOOL;
END_VAR
VAR_OUTPUT
	Error		:	BOOL;
END_VAR
VAR
	Output_Params	:	ARRAY[1..6] OF REAL;
	FirstScan		:	Bool;
END_VAR

        (*Collect Inputs and store them locally*)
Output_Params[1]:=Seconds;
Output_Params[2]:=0;
Output_Params[3]:=0;
Output_Params[4]:=0;
Output_Params[5]:=0;
Output_Params[6]:=0;


(* If Values have change, Reinitialise Outputs*)

IF FirstScan=0 OR Robot.Outputs.MotionCommand.Argument0 <> Output_Params[1] OR Robot.Outputs.MotionCommand.Argument1 <> Output_Params[2] OR Robot.Outputs.MotionCommand.Argument2 <> Output_Params[3] OR Robot.Outputs.MotionCommand.Argument3 <> Output_Params[4] OR Robot.Outputs.MotionCommand.Argument4 <> Output_Params[5] OR Robot.Outputs.MotionCommand.Argument5 <> Output_Params[6] THEN
	Buffered := FALSE;
	Sent := FALSE;
END_IF;

(*if not in legacy mode, Act Setpoint*)
IF Robot.Outputs.MoveID <> 0 THEN
    Robot.Outputs.MotionControl.SetPoint := TRUE;
END_IF;

(* To send _Move, send _Move ID *)
IF NOT Buffered AND NOT Sent THEN
    
    Robot.Outputs.MotionCommand.MoveCommand := Meca500_MotionCommandID.SET_VEL_TIMEOUT;
    Robot.Outputs.MotionCommand.Argument0 := Output_Params[1];
	Robot.Outputs.MotionCommand.Argument1 := Output_Params[2];
	Robot.Outputs.MotionCommand.Argument2 := Output_Params[3];
	Robot.Outputs.MotionCommand.Argument3 := Output_Params[4];
	Robot.Outputs.MotionCommand.Argument4 := Output_Params[5];
	Robot.Outputs.MotionCommand.Argument5 := Output_Params[6];
    
    IF ExternalStateControl THEN
        IF ExternalMoveID <> 0 AND ExternalMoveID <> 32240 AND ExternalMoveID <> 32241 THEN
            Robot.Outputs.MoveID := ExternalMoveID;
            Sent := TRUE;
        END_IF;
        
    ELSE (*Not External Control*)
        IF Robot.Outputs.MoveID = 32240 THEN
            Robot.Outputs.MoveID := 32241;
        ELSIF Robot.Outputs.MoveID = 32241 THEN
            Robot.Outputs.MoveID := 32240;
        ELSIF Robot.Outputs.MoveID <> 32240 OR Robot.Outputs.MoveID <> 32241 THEN
            Robot.Outputs.MoveID := 32240;
        END_IF;
        Sent := TRUE;
    END_IF;
END_IF;

(* Check if _Move has been sent, if so, check if it was received *)
IF Sent THEN
    IF Robot.Outputs.MotionCommand.MoveCommand = Meca500_MotionCommandID.SET_VEL_TIMEOUT THEN
        IF Robot.Outputs.MotionCommand.Argument0 = Output_Params[1] AND Robot.Outputs.MotionCommand.Argument1 = Output_Params[2] AND Robot.Outputs.MotionCommand.Argument2 = Output_Params[3] AND Robot.Outputs.MotionCommand.Argument3 = Output_Params[4] AND Robot.Outputs.MotionCommand.Argument4 = Output_Params[5] AND Robot.Outputs.MotionCommand.Argument5 = Output_Params[6] THEN
            IF Robot.Inputs.Motion.MoveID = Robot.Outputs.MoveID THEN
                Buffered := TRUE;
            END_IF;
        END_IF;
    END_IF;
END_IF;

(*If External _Move ID is equal to Internal, raise an error*)
IF ExternalMoveID = 32240 OR ExternalMoveID = 32241 THEN
    Error := TRUE;
END_IF;
FirstScan:=TRUE;

END_FUNCTION_BLOCK

// Device/Application/F1000_FBs/Meca500/SetWrf
FUNCTION_BLOCK SetWrf
VAR_INPUT
	Pose					:	ARRAY[1..6]OF REAL;
	ExternalStatecontrol 	:	BOOL;
	ExternalMoveID			:	UINT;
END_VAR
VAR_IN_OUT
	Robot	:	Meca500;	
	Sent		:	BOOL;
	Buffered	:	BOOL;
END_VAR
VAR_OUTPUT
	Error		:	BOOL;
END_VAR
VAR
	Output_Params	:	ARRAY[1..6] OF REAL;
	FirstScan		:	BOOL;
END_VAR

        (*Collect Inputs and store them locally*)
Output_Params[1]:=Pose[1];
Output_Params[2]:=Pose[2];
Output_Params[3]:=Pose[3];
Output_Params[4]:=Pose[4];
Output_Params[5]:=Pose[5];
Output_Params[6]:=Pose[6];

(* If Values have change, Reinitialise Outputs*)

IF FirstScan=0 OR Robot.Outputs.MotionCommand.Argument0 <> Output_Params[1] OR Robot.Outputs.MotionCommand.Argument1 <> Output_Params[2] OR Robot.Outputs.MotionCommand.Argument2 <> Output_Params[3] OR Robot.Outputs.MotionCommand.Argument3 <> Output_Params[4] OR Robot.Outputs.MotionCommand.Argument4 <> Output_Params[5] OR Robot.Outputs.MotionCommand.Argument5 <> Output_Params[6] THEN
	Buffered := FALSE;
	Sent := FALSE;
END_IF;

(*if not in legacy mode, Act Setpoint*)
IF Robot.Outputs.MoveID <> 0 THEN
    Robot.Outputs.MotionControl.SetPoint := TRUE;
END_IF;

(* To send _Move, send _Move ID *)
IF NOT Buffered AND NOT Sent THEN
    
    Robot.Outputs.MotionCommand.MoveCommand := Meca500_MotionCommandID.SET_WRF;
    Robot.Outputs.MotionCommand.Argument0 := Output_Params[1];
	Robot.Outputs.MotionCommand.Argument1 := Output_Params[2];
	Robot.Outputs.MotionCommand.Argument2 := Output_Params[3];
	Robot.Outputs.MotionCommand.Argument3 := Output_Params[4];
	Robot.Outputs.MotionCommand.Argument4 := Output_Params[5];
	Robot.Outputs.MotionCommand.Argument5 := Output_Params[6];
    
    IF ExternalStateControl THEN
        IF ExternalMoveID <> 0 AND ExternalMoveID <> 32140 AND ExternalMoveID <> 32141 THEN
            Robot.Outputs.MoveID := ExternalMoveID;
            Sent := TRUE;
        END_IF;
        
    ELSE (*Not External Control*)
        IF Robot.Outputs.MoveID = 32140 THEN
            Robot.Outputs.MoveID := 32141;
        ELSIF Robot.Outputs.MoveID = 32141 THEN
            Robot.Outputs.MoveID := 32140;
        ELSIF Robot.Outputs.MoveID <> 32140 OR Robot.Outputs.MoveID <> 32141 THEN
            Robot.Outputs.MoveID := 32140;
        END_IF;
        Sent := TRUE;
    END_IF;
END_IF;

(* Check if _Move has been sent, if so, check if it was received *)
IF Sent THEN
    IF Robot.Outputs.MotionCommand.MoveCommand = Meca500_MotionCommandID.SET_WRF THEN
        IF Robot.Outputs.MotionCommand.Argument0 = Output_Params[1] AND Robot.Outputs.MotionCommand.Argument1 = Output_Params[2] AND Robot.Outputs.MotionCommand.Argument2 = Output_Params[3] AND Robot.Outputs.MotionCommand.Argument3 = Output_Params[4] AND Robot.Outputs.MotionCommand.Argument4 = Output_Params[5] AND Robot.Outputs.MotionCommand.Argument5 = Output_Params[6] THEN
            IF Robot.Inputs.Motion.MoveID = Robot.Outputs.MoveID THEN
                Buffered := TRUE;
            END_IF;
        END_IF;
    END_IF;
END_IF;

(*If External _Move ID is equal to Internal, raise an error*)
IF ExternalMoveID = 32140 OR ExternalMoveID = 32141 THEN
    Error := TRUE;
END_IF;
FirstScan:=TRUE;

END_FUNCTION_BLOCK

// Device/Application/F1000_FBs/Meca500/StartProgram
FUNCTION_BLOCK StartProgram
VAR_INPUT
	n					:	REAL;
	ExternalStatecontrol 	:	BOOL;
	ExternalMoveID			:	UINT;
END_VAR
VAR_IN_OUT
	Robot	:	Meca500;	
	Sent		:	BOOL;
	Buffered	:	BOOL;
END_VAR
VAR_OUTPUT
	Error		:	BOOL;
END_VAR
VAR
	Output_Params	:	ARRAY[1..6] OF REAL;
	FirstScan		:	Bool;
END_VAR

        (*Collect Inputs and store them locally*)
Output_Params[1]:=n;
Output_Params[2]:=0;
Output_Params[3]:=0;
Output_Params[4]:=0;
Output_Params[5]:=0;
Output_Params[6]:=0;


(* If Values have change, Reinitialise Outputs*)

IF FirstScan=0 OR Robot.Outputs.MotionCommand.Argument0 <> Output_Params[1] OR Robot.Outputs.MotionCommand.Argument1 <> Output_Params[2] OR Robot.Outputs.MotionCommand.Argument2 <> Output_Params[3] OR Robot.Outputs.MotionCommand.Argument3 <> Output_Params[4] OR Robot.Outputs.MotionCommand.Argument4 <> Output_Params[5] OR Robot.Outputs.MotionCommand.Argument5 <> Output_Params[6] THEN
	Buffered := FALSE;
	Sent := FALSE;
END_IF;

(*if not in legacy mode, Act Setpoint*)
IF Robot.Outputs.MoveID <> 0 THEN
    Robot.Outputs.MotionControl.SetPoint := TRUE;
END_IF;

(* To send _Move, send _Move ID *)
IF NOT Buffered AND NOT Sent THEN
    
    Robot.Outputs.MotionCommand.MoveCommand := Meca500_MotionCommandID.START_PROGRAM;
    Robot.Outputs.MotionCommand.Argument0 := Output_Params[1];
	Robot.Outputs.MotionCommand.Argument1 := Output_Params[2];
	Robot.Outputs.MotionCommand.Argument2 := Output_Params[3];
	Robot.Outputs.MotionCommand.Argument3 := Output_Params[4];
	Robot.Outputs.MotionCommand.Argument4 := Output_Params[5];
	Robot.Outputs.MotionCommand.Argument5 := Output_Params[6];
    
    IF ExternalStateControl THEN
        IF ExternalMoveID <> 0 AND ExternalMoveID <> 31900 AND ExternalMoveID <> 31901 THEN
            Robot.Outputs.MoveID := ExternalMoveID;
            Sent := TRUE;
        END_IF;
        
    ELSE (*Not External Control*)
        IF Robot.Outputs.MoveID = 31900 THEN
            Robot.Outputs.MoveID := 31901;
        ELSIF Robot.Outputs.MoveID = 31901 THEN
            Robot.Outputs.MoveID := 31900;
        ELSIF Robot.Outputs.MoveID <> 31900 OR Robot.Outputs.MoveID <> 31901 THEN
            Robot.Outputs.MoveID := 31900;
        END_IF;
        Sent := TRUE;
    END_IF;
END_IF;

(* Check if _Move has been sent, if so, check if it was received *)
IF Sent THEN
    IF Robot.Outputs.MotionCommand.MoveCommand = Meca500_MotionCommandID.START_PROGRAM THEN
        IF Robot.Outputs.MotionCommand.Argument0 = Output_Params[1] AND Robot.Outputs.MotionCommand.Argument1 = Output_Params[2] AND Robot.Outputs.MotionCommand.Argument2 = Output_Params[3] AND Robot.Outputs.MotionCommand.Argument3 = Output_Params[4] AND Robot.Outputs.MotionCommand.Argument4 = Output_Params[5] AND Robot.Outputs.MotionCommand.Argument5 = Output_Params[6] THEN
            IF Robot.Inputs.Motion.MoveID = Robot.Outputs.MoveID THEN
                Buffered := TRUE;
            END_IF;
        END_IF;
    END_IF;
END_IF;

(*If External _Move ID is equal to Internal, raise an error*)
IF ExternalMoveID = 31900 OR ExternalMoveID = 31901 THEN
    Error := TRUE;
END_IF;
FirstScan:=TRUE;

END_FUNCTION_BLOCK

// Device/Application/F020_HMI_Pages/F020_Camera_Robot
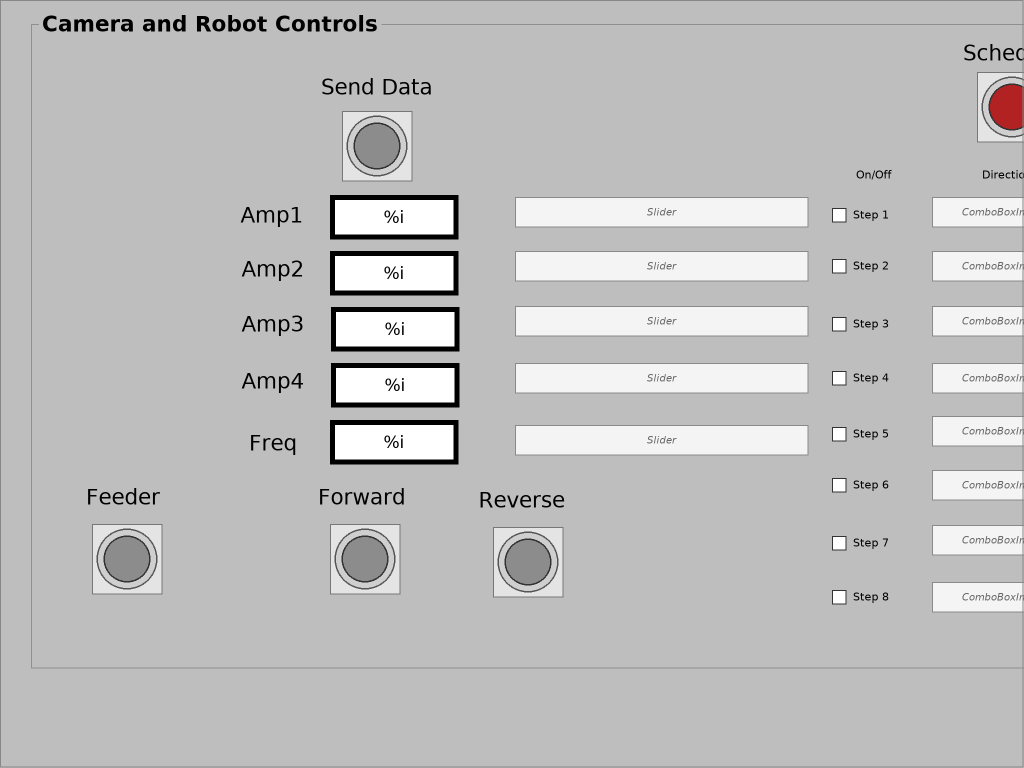
VISUALIZATION F020_Camera_Robot  // 1024x768
    GroupBox (31,16 1221x652), "Camera and Robot Controls"
        Textfield (299,179 128x44), "%i", text variable: GVL.PARTX.Amp1
            OnMouseClick: write the text variable via VisuDialogs.Numpad
        Label (166,184 150x30), "Amp1"
        Textfield (299,235 128x44), "%i", text variable: GVL.PARTX.Amp2
            OnMouseClick: write the text variable via VisuDialogs.Numpad
        Label (167,238 150x30), "Amp2"
        Textfield (300,291 128x44), "%i", text variable: GVL.PARTX.Amp3
            OnMouseClick: write the text variable via VisuDialogs.Numpad
        Label (167,293 150x30), "Amp3"
        Textfield (300,347 128x44), "%i", text variable: GVL.PARTX.Amp4
            OnMouseClick: write the text variable via VisuDialogs.Numpad
        Label (167,350 150x30), "Amp4"
        Textfield (299,404 128x44), "%i", text variable: GVL.PARTX.Freq
            OnMouseClick: write the text variable via VisuDialogs.Numpad
        Label (167,412 150x30), "Freq"
        PushSwitch (61,508 70x70), variable: GVL.PARTX.Feeder_Enable, behaviour: TOGGLE, style: Switch-PushSwitch-Gray
        Label (17,466 150x30), "Feeder"
        Slider (484,181 293x30), variable: GVL.PARTX.Amp1, scale 0..100
        Slider (484,235 293x30), variable: GVL.PARTX.Amp2, scale 0..100
        Slider (484,290 293x30), variable: GVL.PARTX.Amp3, scale 0..100
        Label (256,466 150x30), "Forward"
        Label (472,466 150x30)
        PushSwitch (299,508 70x70), variable: GVL.PARTX.FWD, behaviour: TOGGLE, style: Switch-PushSwitch-Gray
        Label (416,469 150x30), "Reverse"
        PushSwitch (946,56 70x70), variable: GVL.PARTX.SCHED, behaviour: TOGGLE, style: Switch-PushSwitch-Red
        Label (906,22 150x30), "Schedule"
        Checkbox (799,184 150x30), "Step 1", variable: GVL.PARTX.Steps[1].StepEnable
        Checkbox (799,235 150x30), "Step 2", variable: GVL.PARTX.Steps[2].StepEnable
        Checkbox (799,293 150x30), "Step 3", variable: GVL.PARTX.Steps[3].StepEnable
        Checkbox (799,347 150x30), "Step 4", variable: GVL.PARTX.Steps[4].StepEnable
        ComboBoxInteger (901,181 150x30), variable: GVL.PARTX.Steps[1].Direction, text list: 'TL_Directions'
        ComboBoxInteger (901,235 150x30), variable: GVL.PARTX.Steps[2].Direction, text list: 'TL_Directions'
        ComboBoxInteger (901,290 150x30), variable: GVL.PARTX.Steps[3].Direction, text list: 'TL_Directions'
        ComboBoxInteger (901,347 150x30), variable: GVL.PARTX.Steps[4].Direction, text list: 'TL_Directions'
        Textfield (1080,175 128x44), "%i", text variable: GVL.PARTX.Steps[1].DurationMS
            OnMouseClick: write the text variable via VisuDialogs.Numpad
        Checkbox (799,403 150x30), "Step 5", variable: GVL.PARTX.Steps[5].StepEnable
        ComboBoxInteger (901,454 150x30), variable: GVL.PARTX.Steps[6].Direction, text list: 'TL_Directions'
        Label (768,144 150x30), "On/Off"
        Label (901,144 150x30), "Direction"
        Label (1061,144 150x30), "Duration"
        PushSwitch (311,95 70x70), variable: GVL.Explicit.xTriggerWrite, behaviour: TAP, style: Switch-PushSwitch-Gray
        Label (271,56 150x30), "Send Data"
    Slider (515,363 293x30), variable: GVL.PARTX.Amp4, scale 0..100
    Slider (515,425 293x30), variable: GVL.PARTX.Freq, scale 0..100
    PushSwitch (493,527 70x70), variable: GVL.PARTX.REV, behaviour: TOGGLE, style: Switch-PushSwitch-Gray
    Textfield (1111,247 128x44), "%i", text variable: GVL.PARTX.Steps[2].DurationMS
        OnMouseClick: write the text variable via VisuDialogs.Numpad
    Textfield (1112,303 128x44), "%i", text variable: GVL.PARTX.Steps[3].DurationMS
        OnMouseClick: write the text variable via VisuDialogs.Numpad
    Textfield (1112,359 128x44), "%i", text variable: GVL.PARTX.Steps[4].DurationMS
        OnMouseClick: write the text variable via VisuDialogs.Numpad
    Checkbox (830,470 150x30), "Step 6", variable: GVL.PARTX.Steps[6].StepEnable
    Checkbox (830,528 150x30), "Step 7", variable: GVL.PARTX.Steps[7].StepEnable
    Checkbox (830,582 150x30), "Step 8", variable: GVL.PARTX.Steps[8].StepEnable
    ComboBoxInteger (932,416 150x30), variable: GVL.PARTX.Steps[5].Direction, text list: 'TL_Directions'
    ComboBoxInteger (932,525 150x30), variable: GVL.PARTX.Steps[7].Direction, text list: 'TL_Directions'
    ComboBoxInteger (932,582 150x30), variable: GVL.PARTX.Steps[8].Direction, text list: 'TL_Directions'
    Textfield (1111,410 128x44), "%i", text variable: GVL.PARTX.Steps[5].DurationMS
        OnMouseClick: write the text variable via VisuDialogs.Numpad
    Textfield (1111,466 128x44), "%i", text variable: GVL.PARTX.Steps[6].DurationMS
        OnMouseClick: write the text variable via VisuDialogs.Numpad
    Textfield (1112,522 128x44), "%i", text variable: GVL.PARTX.Steps[7].DurationMS
        OnMouseClick: write the text variable via VisuDialogs.Numpad
    Textfield (1112,578 128x44), "%i", text variable: GVL.PARTX.Steps[8].DurationMS
        OnMouseClick: write the text variable via VisuDialogs.Numpad
END_VISUALIZATION

